GLOBALCONSTANTS PgnDef (* Global constants *)
  (* Standard: 61499-1 *)
  (* Version 1.0, 2026-06-29, Franz Höpfinger, Demmler Andreas Fahrzeugbau *)
  PACKAGE isobus::pgn::const;
  VAR_GLOBAL CONSTANT
    PGN_TORQUE_SPEED_CONTROL1 : UDINT := UDINT#16#0000; (* < 00000 - TSC1 *)
    PGN_TRANSMISSION_CONTROL1 : UDINT := UDINT#16#0100; (* < 00256 - TC1 *)
    PGN_ELECTRONIC_BRAKE_SYSTEM_1_1 : UDINT := UDINT#16#0200; (* < 00512 - EBS11 *)
    PGN_ELECTRONIC_BRAKE_SYSTEM_2_1 : UDINT := UDINT#16#0300; (* < 00768 - EBS21 *)
    PGN_EXTERNAL_BRAKE_REQUEST : UDINT := UDINT#16#0400; (* < 01024 - XBR *)
    PGN_CANOPEN_APPLICATION_MESSAGE_1_1 : UDINT := UDINT#16#0500; (* < 01280 - CAM11 *)
    PGN_CANOPEN_APPLICATION_MESSAGE_2_1 : UDINT := UDINT#16#0600; (* < 01536 - CAM21 *)
    PGN_GENERAL_PURPOSE_VALVE_PRESSURE : UDINT := UDINT#16#0700; (* < 01792 - GPV4 *)
    PGN_AUXILIARY_INPUT_OUTPUT_STATUS_5 : UDINT := UDINT#16#0800; (* < 02048 - AUXIO5 *)
    PGN_STATIC_ROLL_ANGLE_SENSOR_INFORMATION : UDINT := UDINT#16#0900; (* < 02304 - SRASI *)
    PGN_CRUISE_CONTROL_VEHICLE_SPEED_2 : UDINT := UDINT#16#0A00; (* < 02560 - CCVS2 *)
    PGN_ADVANCED_EMERGENCY_BRAKING_SYSTEM_2 : UDINT := UDINT#16#0B00; (* < 02816 - AEBS2 *)
    PGN_ELECTRONIC_ENGINE_CONTROLLER_16 : UDINT := UDINT#16#0C00; (* < 03072 - EEC16 *)
    PGN_TRANSMISSION_CONTROL_2 : UDINT := UDINT#16#0D00; (* < 03328 - TC2 *)
    PGN_SAFETY_HEADER_MESSAGE : UDINT := UDINT#16#0E00; (* < 03584 - SHM *)
    PGN_HIGH_VOLTAGE_ENERGY_STORAGE_PACK_11_CONTROL_1 : UDINT := UDINT#16#0F00; (* < 03840 - HVESP11C1 *)
    PGN_HIGH_VOLTAGE_ENERGY_STORAGE_PACK_12_CONTROL_1 : UDINT := UDINT#16#1000; (* < 04096 - HVESP12C1 *)
    PGN_HIGH_VOLTAGE_ENERGY_STORAGE_PACK_13_CONTROL_1 : UDINT := UDINT#16#1100; (* < 04352 - HVESP13C1 *)
    PGN_HIGH_VOLTAGE_ENERGY_STORAGE_PACK_14_CONTROL_1 : UDINT := UDINT#16#1200; (* < 04608 - HVESP14C1 *)
    PGN_HIGH_VOLTAGE_ENERGY_STORAGE_PACK_15_CONTROL_1 : UDINT := UDINT#16#1300; (* < 04864 - HVESP15C1 *)
    PGN_HIGH_VOLTAGE_ENERGY_STORAGE_PACK_16_CONTROL_1 : UDINT := UDINT#16#1400; (* < 05120 - HVESP16C1 *)
    PGN_HIGH_VOLTAGE_ENERGY_STORAGE_PACK_17_CONTROL_1 : UDINT := UDINT#16#1500; (* < 05376 - HVESP17C1 *)
    PGN_HIGH_VOLTAGE_ENERGY_STORAGE_PACK_18_CONTROL_1 : UDINT := UDINT#16#1600; (* < 05632 - HVESP18C1 *)
    PGN_HIGH_VOLTAGE_ENERGY_STORAGE_PACK_19_CONTROL_1 : UDINT := UDINT#16#1700; (* < 05888 - HVESP19C1 *)
    PGN_HIGH_VOLTAGE_ENERGY_STORAGE_PACK_20_CONTROL_1 : UDINT := UDINT#16#1800; (* < 06144 - HVESP20C1 *)
    PGN_HIGH_VOLTAGE_ENERGY_STORAGE_PACK_21_CONTROL_1 : UDINT := UDINT#16#1900; (* < 06400 - HVESP21C1 *)
    PGN_HIGH_VOLTAGE_ENERGY_STORAGE_PACK_22_CONTROL_1 : UDINT := UDINT#16#1A00; (* < 06656 - HVESP22C1 *)
    PGN_HIGH_VOLTAGE_ENERGY_STORAGE_SYSTEM_CONTROL_1 : UDINT := UDINT#16#1B00; (* < 06912 - HVESSC1 *)
    PGN_TRANSMISSION_CONTROL_3_OBSOLETE_SEE_PGN_16896 : UDINT := UDINT#16#1C00; (* < 07168 - TC3 *)
    PGN_ENGINE_IGNITION_CONTROLLER : UDINT := UDINT#16#1D00; (* < 07424 - EIC *)
    PGN_ALTERNATOR_CONTROL : UDINT := UDINT#16#1E00; (* < 07680 - ALTC *)
    PGN_HIGH_VOLTAGE_ENERGY_STORAGE_PACK_23_CONTROL_1 : UDINT := UDINT#16#1F00; (* < 07936 - HVESP23C1 *)
    PGN_HIGH_VOLTAGE_ENERGY_STORAGE_PACK_24_CONTROL_1 : UDINT := UDINT#16#2000; (* < 08192 - HVESP24C1 *)
    PGN_HIGH_VOLTAGE_ENERGY_STORAGE_PACK_25_CONTROL_1 : UDINT := UDINT#16#2100; (* < 08448 - HVESP25C1 *)
    PGN_HIGH_VOLTAGE_ENERGY_STORAGE_PACK_26_CONTROL_1 : UDINT := UDINT#16#2200; (* < 08704 - HVESP26C1 *)
    PGN_TIMS_TO_TIMC : UDINT := UDINT#16#2300; (* < 08960 - TIM12 *)
    PGN_TIMC_TO_TIMS : UDINT := UDINT#16#2400; (* < 09216 - TIM21 *)
    PGN_MULTI_PG : UDINT := UDINT#16#2500; (* < 09472 - MCPG *)
    PGN_MOTOR_GENERATOR_1_INVERTER_CONTROL : UDINT := UDINT#16#2600; (* < 09728 - MG1IC *)
    PGN_MOTOR_GENERATOR_2_INVERTER_CONTROL : UDINT := UDINT#16#2700; (* < 09984 - MG2IC *)
    PGN_MOTOR_GENERATOR_1_INVERTER_RATE_LIMITS_REQUEST_1 : UDINT := UDINT#16#2800; (* < 10240 - MG1IRLR1 *)
    PGN_MOTOR_GENERATOR_2_INVERTER_RATE_LIMITS_REQUEST_1 : UDINT := UDINT#16#2900; (* < 10496 - MG2IRLR1 *)
    PGN_HIGH_VOLTAGE_ENERGY_STORAGE_PACK_1_CONTROL_1 : UDINT := UDINT#16#2A00; (* < 10752 - HVESP1C1 *)
    PGN_HIGH_VOLTAGE_ENERGY_STORAGE_PACK_2_CONTROL_1 : UDINT := UDINT#16#2B00; (* < 11008 - HVESP2C1 *)
    PGN_HIGH_VOLTAGE_ENERGY_STORAGE_PACK_3_CONTROL_1 : UDINT := UDINT#16#2C00; (* < 11264 - HVESP3C1 *)
    PGN_HIGH_VOLTAGE_ENERGY_STORAGE_PACK_4_CONTROL_1 : UDINT := UDINT#16#2D00; (* < 11520 - HVESP4C1 *)
    PGN_HIGH_VOLTAGE_ENERGY_STORAGE_PACK_5_CONTROL_1 : UDINT := UDINT#16#2E00; (* < 11776 - HVESP5C1 *)
    PGN_HIGH_VOLTAGE_ENERGY_STORAGE_PACK_6_CONTROL_1 : UDINT := UDINT#16#2F00; (* < 12032 - HVESP6C1 *)
    PGN_HIGH_VOLTAGE_ENERGY_STORAGE_PACK_7_CONTROL_1 : UDINT := UDINT#16#3000; (* < 12288 - HVESP7C1 *)
    PGN_HIGH_VOLTAGE_ENERGY_STORAGE_PACK_8_CONTROL_1 : UDINT := UDINT#16#3100; (* < 12544 - HVESP8C1 *)
    PGN_HIGH_VOLTAGE_ENERGY_STORAGE_PACK_9_CONTROL_1 : UDINT := UDINT#16#3200; (* < 12800 - HVESP9C1 *)
    PGN_HIGH_VOLTAGE_ENERGY_STORAGE_PACK_10_CONTROL_1 : UDINT := UDINT#16#3300; (* < 13056 - HVESP10C1 *)
    PGN_RELIABLE_LONG_MESSAGE : UDINT := UDINT#16#3400; (* < 13312 - CJLFI *)
    PGN_RELIABLE_SHORT_MESSAGE : UDINT := UDINT#16#3500; (* < 13568 - CJSFWI *)
    PGN_UNRELIABLE_MESSAGE : UDINT := UDINT#16#3600; (* < 13824 - CJSFOI *)
    PGN_MESSAGE_ACKNOWLEDGEMENT : UDINT := UDINT#16#3700; (* < 14080 - CJCFI *)
    PGN_VERSION_NEGOTIATION_SECTION : UDINT := UDINT#16#3800; (* < 14336 - CJVGM *)
    PGN_EXTERNAL_ACC_ACCELERATION_REQUEST : UDINT := UDINT#16#3900; (* < 14592 - XAR *)
    PGN_BATTERY_CHARGER_1_COMMAND_1 : UDINT := UDINT#16#3A00; (* < 14848 - BCH1C1 *)
    PGN_BATTERY_CHARGER_2_COMMAND_1 : UDINT := UDINT#16#3B00; (* < 15104 - BCH2C1 *)
    PGN_TRACTOR_IMPLEMENT_MANAGEMENT_TIM_SERVER_TO_TIM_CLIENT_CONTROL_STATUS : UDINT := UDINT#16#3C00; (* < 15360 - TIM12_CS *)
    PGN_TRACTOR_IMPLEMENT_MANAGEMENT_TIM_CLIENT_TO_TIM_SERVER_CONTROL_STATUS : UDINT := UDINT#16#3D00; (* < 15616 - TIM21_CS *)
    PGN_FUEL_CELL_SYSTEM_CONTROL_COMMAND : UDINT := UDINT#16#3E00; (* < 15872 - FCSCC *)
    PGN_FUEL_CELL_SYSTEM_POWER_LIMIT_COMMAND : UDINT := UDINT#16#3F00; (* < 16128 - FCSPLC *)
    PGN_FUEL_CELL_SYSTEM_CURRENT_LIMIT_COMMAND : UDINT := UDINT#16#4000; (* < 16384 - FCSCLC *)
    PGN_HYDROGEN_STORAGE_SYSTEM_CONTROL_COMMAND : UDINT := UDINT#16#4100; (* < 16640 - HSSCC *)
    PGN_TRANSMISSION_CONTROL_4 : UDINT := UDINT#16#4200; (* < 16896 - TC4 *)
    PGN_SAFETY_HEADER_MESSAGE_2 : UDINT := UDINT#16#4300; (* < 17152 - SHM2 *)
    PGN_API_SELECT : UDINT := UDINT#16#4600; (* < 17920 - APISEL *)
    PGN_TRACTOR_IMPLEMENT_MANAGEMENT_TIM_SERVER_TO_CLIENT_INITIALIZATION_PARAMETE_X : UDINT := UDINT#16#4800; (* < 18432 - TIM12_IP *)
    PGN_TRACTOR_IMPLEMENT_MANAGEMENT_TIM_CLIENT_TO_SERVER_INITIALIZATION_PARAMETE_X : UDINT := UDINT#16#4900; (* < 18688 - TIM21_IP *)
    PGN_EV_MULTI_CONNECTION_DC_STATUS_1 : UDINT := UDINT#16#4A00; (* < 18944 - EVMCDCS1 *)
    PGN_EV_MULTI_CONNECTION_DC_CHARGING_LIMITS_1 : UDINT := UDINT#16#4B00; (* < 19200 - EVMCDCLIM1 *)
    PGN_ELECTRIFIED_ACCESSORY_ENGINE_COOLANT_PUMP_COMMAND : UDINT := UDINT#16#4C00; (* < 19456 - EAECPC *)
    PGN_FD_TRANSPORT_PROTOCOL_CONNECTION_MGMT : UDINT := UDINT#16#4D00; (* < 19712 - FD.TP.CM *)
    PGN_FD_TRANSPORT_PROTOCOL_DATA_TRANSFER : UDINT := UDINT#16#4E00; (* < 19968 - FD.TP.DT *)
    PGN_DATA_TRANSFER_SUPPORT : UDINT := UDINT#16#4F00; (* < 20224 - DTS *)
    PGN_MONTHLY_DATA_TRANSFER : UDINT := UDINT#16#5000; (* < 20480 - MDT *)
    PGN_WEEKLY_DATA_TRANSFER : UDINT := UDINT#16#5100; (* < 20736 - WDT *)
    PGN_DAILY_DATA_TRANSFER : UDINT := UDINT#16#5200; (* < 20992 - DDT *)
    PGN_EVSE_CONTROL_1 : UDINT := UDINT#16#5300; (* < 21248 - EVSEC1 *)
    PGN_WINCH_INFORMATION_3 : UDINT := UDINT#16#5400; (* < 21504 - WINCH3 *)
    PGN_AIR_SUSPENSION_CONTROL_8 : UDINT := UDINT#16#5500; (* < 21760 - ASC8 *)
    PGN_MOTOR_GENERATOR_2_INVERTER_CONTROL_2 : UDINT := UDINT#16#5600; (* < 22016 - MG2IC2 *)
    PGN_MOTOR_GENERATOR_1_INVERTER_CONTROL_2 : UDINT := UDINT#16#5700; (* < 22272 - MG1IC2 *)
    PGN_HOIST_COMMAND_INFORMATION : UDINT := UDINT#16#5800; (* < 22528 - HCI2 *)
    PGN_MOTOR_GENERATOR_2_INVERTER_ISOLATION_INTEGRITY_REQUEST : UDINT := UDINT#16#5900; (* < 22784 - MG2IIR *)
    PGN_MOTOR_GENERATOR_1_INVERTER_ISOLATION_INTEGRITY_REQUEST : UDINT := UDINT#16#5A00; (* < 23040 - MG1IIR *)
    PGN_MOTOR_GENERATOR_2_INVERTER_LIMITS_REQUEST_POWER : UDINT := UDINT#16#5B00; (* < 23296 - MG2IRP *)
    PGN_MOTOR_GENERATOR_2_INVERTER_LIMITS_REQUEST_MECHANICAL : UDINT := UDINT#16#5C00; (* < 23552 - MG2ILRM *)
    PGN_MOTOR_GENERATOR_2_INVERTER_LIMITS_REQUEST_DC_SIDE : UDINT := UDINT#16#5D00; (* < 23808 - MG2ILRDC *)
    PGN_MOTOR_GENERATOR_1_INVERTER_LIMITS_REQUEST_DC_SIDE : UDINT := UDINT#16#5E00; (* < 24064 - MG1ILRDC *)
    PGN_MOTOR_GENERATOR_1_INVERTER_LIMITS_REQUEST_MECHANICAL : UDINT := UDINT#16#5F00; (* < 24320 - MG1ILRM *)
    PGN_MOTOR_GENERATOR_1_INVERTER_LIMITS_REQUEST_POWER : UDINT := UDINT#16#6000; (* < 24576 - MG1IRP *)
    PGN_PERSONNEL_DETECT_INTERLOCK : UDINT := UDINT#16#6100; (* < 24832 - PDI *)
    PGN_ENGINE_CYLINDER_COMBUSTION_CONFIGURATION_FEEDBACK : UDINT := UDINT#16#6200; (* < 25088 - ECCCF *)
    PGN_ENGINE_CYLINDER_COMBUSTION_CONFIGURATION : UDINT := UDINT#16#6300; (* < 25344 - ECCC *)
    PGN_ENGINE_CYLINDER_PRESSURE_TIMING_FEEDBACK : UDINT := UDINT#16#6400; (* < 25600 - ECPTF *)
    PGN_ENGINE_CYLINDER_PRESSURE_TIMING_CONFIGURATION : UDINT := UDINT#16#6500; (* < 25856 - ECPTC *)
    PGN_ELECTRIFIED_ACCESSORY_GENERATOR_COOLANT_PUMP_COMMAND : UDINT := UDINT#16#6600; (* < 26112 - EAGCPC *)
    PGN_ELECTRIFIED_ACCESSORY_GENERATOR_COOLANT_FAN_COMMAND : UDINT := UDINT#16#6700; (* < 26368 - EAGCFC *)
    PGN_ON_BOARD_PROGRAMMING_1 : UDINT := UDINT#16#6800; (* < 26624 - OBP1 *)
    PGN_MARINE_CONTROL_INFORMATION_CONFIGURATION_1 : UDINT := UDINT#16#6900; (* < 26880 - MCIC1 *)
    PGN_MARINE_CONTROL_INFORMATION_2 : UDINT := UDINT#16#6A00; (* < 27136 - MCI2 *)
    PGN_WELL_STIMULATION_PUMP_SENSOR_CALIBRATION_COMMAND : UDINT := UDINT#16#6B00; (* < 27392 - WSPSCC *)
    PGN_CIA_602_2_XCP_OBSOLETE : UDINT := UDINT#16#6C00; (* < 27648 - CXCP *)
    PGN_WELL_STIMULATION_PUMP_SYSTEM_CONFIGURATION_COMMAND : UDINT := UDINT#16#6D00; (* < 27904 - WSPT1 *)
    PGN_CONFIGURABLE_RECEIVE_SPNS_COMMAND : UDINT := UDINT#16#6E00; (* < 28160 - CRSC *)
    PGN_AUTC_TO_AUTS : UDINT := UDINT#16#6F00; (* < 28416 - AUTH21 *)
    PGN_AUTS_TO_AUTC : UDINT := UDINT#16#7000; (* < 28672 - AUTH12 *)
    PGN_CONFIGURABLE_TRANSMIT_PGNS_COMMAND : UDINT := UDINT#16#7100; (* < 28928 - CTPC *)
    PGN_OIL_DEBRIS_MONITOR_CONFIGURATION_COMMAND : UDINT := UDINT#16#7200; (* < 29184 - ODMCC *)
    PGN_ELECTRIFIED_ACCESSORY_PROPULSION_MOTOR_COOLANT_FAN_3_COMMAND : UDINT := UDINT#16#7300; (* < 29440 - EAPMCF3C *)
    PGN_ELECTRIFIED_ACCESSORY_PROPULSION_MOTOR_COOLANT_FAN_2_COMMAND : UDINT := UDINT#16#7400; (* < 29696 - EAPMCF2C *)
    PGN_ELECTRIFIED_ACCESSORY_PROPULSION_MOTOR_COOLANT_FAN_1_COMMAND : UDINT := UDINT#16#7500; (* < 29952 - EAPMCF1C *)
    PGN_ELECTRIFIED_ACCESSORY_POWER_ELECTRONICS_COOLANT_FAN_3_COMMAND : UDINT := UDINT#16#7600; (* < 30208 - EAPECF3C *)
    PGN_ELECTRIFIED_ACCESSORY_POWER_ELECTRONICS_COOLANT_FAN_2_COMMAND : UDINT := UDINT#16#7700; (* < 30464 - EAPECF2C *)
    PGN_ELECTRIFIED_ACCESSORY_POWER_ELECTRONICS_COOLANT_FAN_1_COMMAND : UDINT := UDINT#16#7800; (* < 30720 - EAPECF1C *)
    PGN_ELECTRIFIED_ACCESSORY_PROPULSION_MOTOR_OIL_PUMP_COMMAND : UDINT := UDINT#16#7900; (* < 30976 - EAPMOPC *)
    PGN_ELECTRIFIED_ACCESSORY_PROPULSION_MOTOR_COOLANT_PUMP_COMMAND : UDINT := UDINT#16#7A00; (* < 31232 - EAPMCPC *)
    PGN_ELECTRIFIED_ACCESSORY_POWER_ELECTRONICS_COOLANT_PUMP_COMMAND : UDINT := UDINT#16#7B00; (* < 31488 - EAPECPC *)
    PGN_EXTENDED_CONTROL_FUNCTION_FUNCTIONALITIES : UDINT := UDINT#16#7C00; (* < 31744 - ECFF *)
    PGN_ELECTRIFIED_ACCESSORY_MOTOR_COMMAND : UDINT := UDINT#16#7D00; (* < 32000 - EAMC *)
    PGN_ENGINE_SPEED_RAMP_RATE_BOUNDARY_REQUEST : UDINT := UDINT#16#7E00; (* < 32256 - ESRRBR *)
    PGN_TIRE_SENSOR_IDENTIFICATION_COMMAND : UDINT := UDINT#16#7F00; (* < 32512 - TSIC *)
    PGN_HYBRID_OR_EV_SYSTEM_CONTROL_1 : UDINT := UDINT#16#8000; (* < 32768 - HSC1 *)
    PGN_AFTERTREATMENT_SYSTEM_CONTROL : UDINT := UDINT#16#8100; (* < 33024 - AFTSC *)
    PGN_TIRE_CONFIGURATION_COMMAND_INFORMATION : UDINT := UDINT#16#8200; (* < 33280 - TCCI *)
    PGN_PAYLOAD_CALIBRATION_INFORMATION_COMMAND : UDINT := UDINT#16#8300; (* < 33536 - PCIC *)
    PGN_AFTERTREATMENT_1_PARTICULATE_SENSOR_CONTROL : UDINT := UDINT#16#8400; (* < 33792 - AFT1PSC *)
    PGN_CAB_MESSAGE_2 : UDINT := UDINT#16#8500; (* < 34048 - CM2 *)
    PGN_SWITCHED_POWER_OUTPUTS_COMMAND : UDINT := UDINT#16#8600; (* < 34304 - SPOC *)
    PGN_ENGINE_STATE_REQUESTS : UDINT := UDINT#16#8700; (* < 34560 - ESR *)
    PGN_RADIO_BEACON_REQUEST : UDINT := UDINT#16#8800; (* < 34816 - RBR *)
    PGN_RUNNING_GEAR_EQUIPMENT_2_4 : UDINT := UDINT#16#8900; (* < 35072 - RGE24 *)
    PGN_RUNNING_GEAR_EQUIPMENT_1_2 : UDINT := UDINT#16#8A00; (* < 35328 - RGE12 *)
    PGN_CCP_DATA_TRANSMISSION_OBJECT : UDINT := UDINT#16#8B00; (* < 35584 - CCP_DTO *)
    PGN_CCP_COMMAND_RECEIVE_OBJECT : UDINT := UDINT#16#8C00; (* < 35840 - CCP_CRO *)
    PGN_SCC_TO_SCM : UDINT := UDINT#16#8D00; (* < 36096 - SCCCM *)
    PGN_SCM_TO_SCC : UDINT := UDINT#16#8E00; (* < 36352 - SCMCC *)
    PGN_ENGINE_CONFIGURATION_COMMANDS : UDINT := UDINT#16#8F00; (* < 36608 - ECC *)
    PGN_SUPPLEMENTAL_FAN_COMMAND : UDINT := UDINT#16#9000; (* < 36864 - SFC *)
    PGN_VEHICLE_CHASSIS_LUBRICATION_SYSTEM_1 : UDINT := UDINT#16#9100; (* < 37120 - VLS1 *)
    PGN_AFTERTREATMENT_1_HYDROCARBON_DOSER_INFORMATION_1 : UDINT := UDINT#16#9200; (* < 37376 - HCDI1 *)
    PGN_NAME_MANAGEMENT : UDINT := UDINT#16#9300; (* < 37632 - NM *)
    PGN_AFTERTREATMENT_1_DIESEL_PARTICULATE_FILTER_SOOT_SENSOR_CALIBRATION : UDINT := UDINT#16#9400; (* < 37888 - AT1DPFSSC *)
    PGN_AFTERTREATMENT_2_DIESEL_PARTICULATE_FILTER_SOOT_SENSOR_CALIBRATION : UDINT := UDINT#16#9500; (* < 38144 - AT2DPFSSC *)
    PGN_LOW_VOLTAGE_DISCONNECT_SET_OPERATING_MODE : UDINT := UDINT#16#9600; (* < 38400 - LVDSOM *)
    PGN_NOISE_CONTROL_STATUS : UDINT := UDINT#16#9700; (* < 38656 - NCS *)
    PGN_NOISE_CONTROL_1 : UDINT := UDINT#16#9800; (* < 38912 - NC1 *)
    PGN_JOYSTICK_LAMP_COMMAND_MESSAGE : UDINT := UDINT#16#9900; (* < 39168 - JLCM *)
    PGN_GENERAL_PURPOSE_MESSAGE_1_8 : UDINT := UDINT#16#9A00; (* < 39424 - GPM18 *)
    PGN_PROPRIETARY_METHOD_IDENTIFICATION : UDINT := UDINT#16#9B00; (* < 39680 - PMI *)
    PGN_AUXILIARY_INPUT_OUTPUT_STATUS_7 : UDINT := UDINT#16#9C00; (* < 39936 - AUXIO7 *)
    PGN_AUXILIARY_INPUT_OUTPUT_STATUS_6 : UDINT := UDINT#16#9D00; (* < 40192 - AUXIO6 *)
    PGN_DTC_COUNTS : UDINT := UDINT#16#9E00; (* < 40448 - DM29 *)
    PGN_IMMEDIATE_FAULT_STATUS : UDINT := UDINT#16#9F00; (* < 40704 - DM35 *)
    PGN_NTE_STATUS : UDINT := UDINT#16#A000; (* < 40960 - DM34 *)
    PGN_EMISSION_INCREASING_AUXILIARY_EMISSION_CONTROL_DEVICE_ACTIVE_TIME : UDINT := UDINT#16#A100; (* < 41216 - DM33 *)
    PGN_REGULATED_EXHAUST_EMISSION_LEVEL_EXCEEDANCE : UDINT := UDINT#16#A200; (* < 41472 - DM32 *)
    PGN_DTC_TO_LAMP_ASSOCIATION : UDINT := UDINT#16#A300; (* < 41728 - DM31 *)
    PGN_SCALED_TEST_RESULTS : UDINT := UDINT#16#A400; (* < 41984 - DM30 *)
    PGN_AUXILIARY_INPUT_OUTPUT_STATUS_4 : UDINT := UDINT#16#A500; (* < 42240 - AUXIO4 *)
    PGN_AUXILIARY_INPUT_OUTPUT_STATUS_3 : UDINT := UDINT#16#A600; (* < 42496 - AUXIO3 *)
    PGN_AUX_IO_STATUS_2 : UDINT := UDINT#16#A700; (* < 42752 - AUXIO2 *)
    PGN_TEXT_DISPLAY : UDINT := UDINT#16#A800; (* < 43008 - DISP1 *)
    PGN_FORWARD_LANE_IMAGE_COMMAND : UDINT := UDINT#16#A900; (* < 43264 - FLIC *)
    PGN_FSC_TO_FS : UDINT := UDINT#16#AA00; (* < 43520 - CFS *)
    PGN_FS_TO_FSC : UDINT := UDINT#16#AB00; (* < 43776 - FSC *)
    PGN_GUIDANCE_MACHINE_STATUS : UDINT := UDINT#16#AC00; (* < 44032 - GMS *)
    PGN_GUIDANCE_SYSTEM_COMMAND_MSG : UDINT := UDINT#16#AD00; (* < 44288 - GSC *)
    PGN_TIRE_PRESSURE_REFERENCE_SETTING : UDINT := UDINT#16#AE00; (* < 44544 - TPRS *)
    PGN_PARAMETER_LOCATE_MESSAGE : UDINT := UDINT#16#AF00; (* < 44800 - PLM *)
    PGN_CONFIGURATION_IDENTIFICATION_MESSAGE : UDINT := UDINT#16#B000; (* < 45056 - CIM *)
    PGN_PROPRIETARILY_CONFIGURABLE_MESSAGE_1 : UDINT := UDINT#16#B100; (* < 45312 - PCM1 *)
    PGN_PROPRIETARILY_CONFIGURABLE_MESSAGE_2 : UDINT := UDINT#16#B200; (* < 45568 - PCM2 *)
    PGN_PROPRIETARILY_CONFIGURABLE_MESSAGE_3 : UDINT := UDINT#16#B300; (* < 45824 - PCM3 *)
    PGN_PROPRIETARILY_CONFIGURABLE_MESSAGE_4 : UDINT := UDINT#16#B400; (* < 46080 - PCM4 *)
    PGN_PROPRIETARILY_CONFIGURABLE_MESSAGE_5 : UDINT := UDINT#16#B500; (* < 46336 - PCM5 *)
    PGN_PROPRIETARILY_CONFIGURABLE_MESSAGE_6 : UDINT := UDINT#16#B600; (* < 46592 - PCM6 *)
    PGN_PROPRIETARILY_CONFIGURABLE_MESSAGE_7 : UDINT := UDINT#16#B700; (* < 46848 - PCM7 *)
    PGN_PROPRIETARILY_CONFIGURABLE_MESSAGE_8 : UDINT := UDINT#16#B800; (* < 47104 - PCM8 *)
    PGN_PROPRIETARILY_CONFIGURABLE_MESSAGE_9 : UDINT := UDINT#16#B900; (* < 47360 - PCM9 *)
    PGN_PROPRIETARILY_CONFIGURABLE_MESSAGE_10 : UDINT := UDINT#16#BA00; (* < 47616 - PCM10 *)
    PGN_PROPRIETARILY_CONFIGURABLE_MESSAGE_11 : UDINT := UDINT#16#BB00; (* < 47872 - PCM11 *)
    PGN_PROPRIETARILY_CONFIGURABLE_MESSAGE_12 : UDINT := UDINT#16#BC00; (* < 48128 - PCM12 *)
    PGN_PROPRIETARILY_CONFIGURABLE_MESSAGE_13 : UDINT := UDINT#16#BD00; (* < 48384 - PCM13 *)
    PGN_PROPRIETARILY_CONFIGURABLE_MESSAGE_14 : UDINT := UDINT#16#BE00; (* < 48640 - PCM14 *)
    PGN_PROPRIETARILY_CONFIGURABLE_MESSAGE_15 : UDINT := UDINT#16#BF00; (* < 48896 - PCM15 *)
    PGN_PROPRIETARILY_CONFIGURABLE_MESSAGE_16 : UDINT := UDINT#16#C000; (* < 49152 - PCM16 *)
    PGN_DIAGNOSTIC_READINESS_2 : UDINT := UDINT#16#C100; (* < 49408 - DM21 *)
    PGN_MONITOR_PERFORMANCE_RATIO : UDINT := UDINT#16#C200; (* < 49664 - DM20 *)
    PGN_INDIVIDUAL_CLEAR_RESET_OF_ACTIVE_AND_PREVIOUSLY_ACTIVE_DTC : UDINT := UDINT#16#C300; (* < 49920 - DM22 *)
    PGN_GENPURPOSE_VALVE_COMMAND : UDINT := UDINT#16#C400; (* < 50176 - GPV3 *)
    PGN_GENPURPOSE_VALVE_MEASFLOW : UDINT := UDINT#16#C500; (* < 50432 - GPV2 *)
    PGN_GENPURPOSE_VALVE_ESTIMFLOW : UDINT := UDINT#16#C600; (* < 50688 - GPV1 *)
    PGN_ETP_DT : UDINT := UDINT#16#C700; (* < 50944 - ETP.DT *)
    PGN_ETP_CM : UDINT := UDINT#16#C800; (* < 51200 - ETP.CM *)
    PGN_REQUEST2_PGN : UDINT := UDINT#16#C900; (* < 51456 - RQST2 *)
    PGN_TRANSFER_PGN : UDINT := UDINT#16#CA00; (* < 51712 - XFER *)
    PGN_PROCESS_DATA : UDINT := UDINT#16#CB00; (* < 51968 - PD *)
    PGN_REQ_FOR_REP_RATE : UDINT := UDINT#16#CC00; (* < 52224 - REQRR *)
    PGN_DoCAN_MIXED_FUNCTIONAL : UDINT := UDINT#16#CD00; (* < 52480 - DIAG1 *)
    PGN_DoCAN_MIXED_PHYSICAL : UDINT := UDINT#16#CE00; (* < 52736 - DIAG2 *)
    PGN_CONTINUOUSTORQUE : UDINT := UDINT#16#CF00; (* < 52992 - CTL *)
    PGN_CAB_ILLUMINATION : UDINT := UDINT#16#D000; (* < 53248 - CL *)
    PGN_AIRSUSPENSION_CONTROL6 : UDINT := UDINT#16#D100; (* < 53504 - ASC6 *)
    PGN_AIRSUSPENSION_CONTROL2 : UDINT := UDINT#16#D200; (* < 53760 - ASC2 *)
    PGN_CALIBRATION_INFORMATION : UDINT := UDINT#16#D300; (* < 54016 - DM19 *)
    PGN_DATA_SECURITY_54272 : UDINT := UDINT#16#D400; (* < 54272 - DM18 *)
    PGN_DATA_SECURITY : UDINT := UDINT#16#D500; (* < 54528 - TDA *)
    PGN_BOOT_LOAD_DATA : UDINT := UDINT#16#D600; (* < 54784 - DM17 *)
    PGN_BINARY_DATA_TRANSFER : UDINT := UDINT#16#D700; (* < 55040 - DM16 *)
    PGN_MEMORY_ACCESS_RESPONSE : UDINT := UDINT#16#D800; (* < 55296 - DM15 *)
    PGN_MEMORY_ACCESS_REQUEST : UDINT := UDINT#16#D900; (* < 55552 - DM14 *)
    PGN_DoCAN_NORMAL_PHYSICAL : UDINT := UDINT#16#DA00; (* < 55808 - DIAG3 *)
    PGN_DoCAN_NORMAL_FUNCTIONAL : UDINT := UDINT#16#DB00; (* < 56064 - DIAG4 *)
    PGN_ANTI_SHEFT_STATUS : UDINT := UDINT#16#DC00; (* < 56320 - ATS *)
    PGN_ANTI_SHEFT_REQUEST : UDINT := UDINT#16#DD00; (* < 56576 - ATR *)
    PGN_RESET : UDINT := UDINT#16#DE00; (* < 56832 - RESET *)
    PGN_STOP_START_BROADCAST : UDINT := UDINT#16#DF00; (* < 57088 - DM13 *)
    PGN_CAB_MESSAGE1 : UDINT := UDINT#16#E000; (* < 57344 - CM1 *)
    PGN_GENERAL_PURPOSE_MESSAGE_2_1 : UDINT := UDINT#16#E100; (* < 57600 - GPM21 *)
    PGN_GENERAL_PURPOSE_MESSAGE_1_1 : UDINT := UDINT#16#E200; (* < 57856 - GPM11 *)
    PGN_CMD_NONCONTIN_MONITOR : UDINT := UDINT#16#E300; (* < 58112 - DM7 *)
    PGN_RUNNING_GEAR_EQUIPMENT_1_1 : UDINT := UDINT#16#E400; (* < 58368 - RGE11 *)
    PGN_RUNNING_GEAR_EQUIPMENT_2_1 : UDINT := UDINT#16#E500; (* < 58624 - RGE21 *)
    PGN_VTtoECU : UDINT := UDINT#16#E600; (* < 58880 - VT12 *)
    PGN_ECUtoVT : UDINT := UDINT#16#E700; (* < 59136 - VT21 *)
    PGN_N_ACK : UDINT := UDINT#16#E800; (* < 59392 - ACKM *)
    PGN_REQUEST_PGN : UDINT := UDINT#16#EA00; (* < 59904 - RQST *)
    PGN_TP_DT : UDINT := UDINT#16#EB00; (* < 60160 - TP.DT *)
    PGN_TP_CM : UDINT := UDINT#16#EC00; (* < 60416 - TP.CM.xx *)
    PGN_NETWORK_LAYER : UDINT := UDINT#16#ED00; (* < 60672 - N.xx *)
    PGN_ADDRESS_CLAIMED : UDINT := UDINT#16#EE00; (* < 60928 - AC *)
    PGN_CANNOT_CLAIM_SA : UDINT := UDINT#16#EE00; (* < 60928 - AC *)
    PGN_PDU1_PropA : UDINT := UDINT#16#EF00; (* < 61184 - PropA *)
    PGN_PDU2_240_X : UDINT := UDINT#16#F000; (* < 61440 - ERC1 *)
    PGN_ELEC_RETARDER_CONTROLLER : UDINT := UDINT#16#F000; (* < 61440 - ERC1 *)
    PGN_ELEC_BRAKE_CONTROLLER : UDINT := UDINT#16#F001; (* < 61441 - EBC1 *)
    PGN_ELEC_TRANSMISS_CONTROLLER_1 : UDINT := UDINT#16#F002; (* < 61442 - ETC1 *)
    PGN_ELEC_ENGINE_CONTROLLER_2 : UDINT := UDINT#16#F003; (* < 61443 - EEC2 *)
    PGN_ELEC_ENGINE_CONTROLLER_1 : UDINT := UDINT#16#F004; (* < 61444 - EEC1 *)
    PGN_ELEC_TRANSMISS_CONTROLLER_2 : UDINT := UDINT#16#F005; (* < 61445 - ETC2 *)
    PGN_ELEC_AXLE_CONTROLLER_1 : UDINT := UDINT#16#F006; (* < 61446 - EAC1 *)
    PGN_FORW_LANE_IMAGE_URGENT_MSG : UDINT := UDINT#16#F007; (* < 61447 - FLI1 *)
    PGN_HYDRAULIC_PRESS_GOVER_INFO : UDINT := UDINT#16#F008; (* < 61448 - HPG *)
    PGN_VEHICLE_DYN_STAB_CTRL_2 : UDINT := UDINT#16#F009; (* < 61449 - VDC2 *)
    PGN_ENGINE_GAS_FLOW_RATE : UDINT := UDINT#16#F00A; (* < 61450 - EGF1 *)
    PGN_ELECTRONIC_STEERING_CONTROL : UDINT := UDINT#16#F00B; (* < 61451 - ESC1 *)
    PGN_ELECTRONIC_TRANSMISSION_CONTROLLER_8 : UDINT := UDINT#16#F00C; (* < 61452 - ETC8 *)
    PGN_LAND_LEVELING_SYSTEM_OPERATIONAL_INFORMATION : UDINT := UDINT#16#F00D; (* < 61453 - LOI *)
    PGN_AFTERTREATMENT_1_INTAKE_GAS_1 : UDINT := UDINT#16#F00E; (* < 61454 - AT1IG1 *)
    PGN_AFTERTREATMENT_1_OUTLET_GAS_1 : UDINT := UDINT#16#F00F; (* < 61455 - AT1OG1 *)
    PGN_AFTERTREATMENT_2_INTAKE_GAS_1 : UDINT := UDINT#16#F010; (* < 61456 - AT2IG1 *)
    PGN_AFTERTREATMENT_2_OUTLET_GAS_1 : UDINT := UDINT#16#F011; (* < 61457 - AT2OG1 *)
    PGN_FIFTH_WHEEL_SMART_SYSTEMS_1 : UDINT := UDINT#16#F012; (* < 61458 - FWSS1 *)
    PGN_SLOPE_SENSOR_INFORMATION : UDINT := UDINT#16#F013; (* < 61459 - SSI *)
    PGN_BLADE_INFORMATION : UDINT := UDINT#16#F014; (* < 61460 - BI *)
    PGN_REQUESTED_GENERATOR_TOTAL_AC_REACTIVE_POWER : UDINT := UDINT#16#F015; (* < 61461 - RGTACRP *)
    PGN_CYLINDER_COMBUSTION_STATUS : UDINT := UDINT#16#F016; (* < 61462 - CCS *)
    PGN_ENGINE_KNOCK_LEVEL_1 : UDINT := UDINT#16#F017; (* < 61463 - KL1 *)
    PGN_ENGINE_KNOCK_LEVEL_2 : UDINT := UDINT#16#F018; (* < 61464 - KL2 *)
    PGN_ENGINE_KNOCK_LEVEL_3 : UDINT := UDINT#16#F019; (* < 61465 - KL3 *)
    PGN_ENGINE_THROTTLE_FUEL_ACTUATOR_CONTROL_COMMAND : UDINT := UDINT#16#F01A; (* < 61466 - TFAC *)
    PGN_GENERAL_PURPOSE_MESSAGE_1_7 : UDINT := UDINT#16#F01B; (* < 61467 - GPM17 *)
    PGN_REQUESTED_GENERATOR_AVERAGE_BASIC_AC_QUANTITIES : UDINT := UDINT#16#F01C; (* < 61468 - RGAAC *)
    PGN_STEERING_ANGLE_SENSOR_INFORMATION : UDINT := UDINT#16#F01D; (* < 61469 - SAS *)
    PGN_GENERATOR_CONTROL_2 : UDINT := UDINT#16#F01E; (* < 61470 - GC2 *)
    PGN_ELECTRONIC_BRAKE_SYSTEM_2_6 : UDINT := UDINT#16#F01F; (* < 61471 - EBS26 *)
    PGN_ELECTRONIC_BRAKE_SYSTEM_2_5 : UDINT := UDINT#16#F020; (* < 61472 - EBS25 *)
    PGN_ENGINE_SPEED_SENSOR_INFORMATION_1 : UDINT := UDINT#16#F021; (* < 61473 - ESSI1 *)
    PGN_MACHINE_SELECTED_SPEED : UDINT := UDINT#16#F022; (* < 61474 - MSS *)
    PGN_AFTERTREATMENT_1_SCR_DOSING_SYSTEM_INFORMATION_1 : UDINT := UDINT#16#F023; (* < 61475 - A1SCRDSI1 *)
    PGN_AFTERTREATMENT_1_SCR_DOSING_SYSTEM_REQUESTS_1 : UDINT := UDINT#16#F024; (* < 61476 - A1SCRDSR1 *)
    PGN_AFTERTREATMENT_1_SCR_AMMONIA_INFORMATION : UDINT := UDINT#16#F025; (* < 61477 - A1SCRAI *)
    PGN_AFTERTREATMENT_2_SCR_DOSING_SYSTEM_INFORMATION_1 : UDINT := UDINT#16#F026; (* < 61478 - A2SCRDSI1 *)
    PGN_AFTERTREATMENT_2_SCR_DOSING_SYSTEM_REQUESTS_1 : UDINT := UDINT#16#F027; (* < 61479 - A2SCRDSR1 *)
    PGN_AFTERTREATMENT_2_SCR_AMMONIA_INFORMATION : UDINT := UDINT#16#F028; (* < 61480 - A2SCRAI *)
    PGN_SLOPE_SENSOR_INFORMATION_2 : UDINT := UDINT#16#F029; (* < 61481 - SSI2 *)
    PGN_ANGULAR_RATE_INFORMATION : UDINT := UDINT#16#F02A; (* < 61482 - ARI *)
    PGN_CRASH_NOTIFICATION : UDINT := UDINT#16#F02B; (* < 61483 - CN *)
    PGN_MAGNET_STATUS_INFORMATION_2 : UDINT := UDINT#16#F02C; (* < 61484 - MSI2 *)
    PGN_ACCELERATION_SENSOR : UDINT := UDINT#16#F02D; (* < 61485 - ACCS *)
    PGN_ENGINE_TURBOCHARGER_CONTROL_1 : UDINT := UDINT#16#F02E; (* < 61486 - ETCC1 *)
    PGN_ADVANCED_EMERGENCY_BRAKING_SYSTEM_1 : UDINT := UDINT#16#F02F; (* < 61487 - AEBS1 *)
    PGN_WIRELESS_STATUS : UDINT := UDINT#16#F030; (* < 61488 - WS *)
    PGN_WAND_SENSOR : UDINT := UDINT#16#F031; (* < 61489 - WAND *)
    PGN_LINEAR_DISPLACEMENT_SENSOR : UDINT := UDINT#16#F032; (* < 61490 - LDISP *)
    PGN_AFTERTREATMENT_1_SCR_AMMONIA_INFORMATION_2 : UDINT := UDINT#16#F033; (* < 61491 - A1SCRAI2 *)
    PGN_AFTERTREATMENT_2_SCR_AMMONIA_INFORMATION_2 : UDINT := UDINT#16#F034; (* < 61492 - A2SCRAI2 *)
    PGN_HIGH_VOLTAGE_ENERGY_STORAGE_SYSTEM_STATUS_2 : UDINT := UDINT#16#F036; (* < 61494 - HVESSS2 *)
    PGN_ENGINE_TURBOCHARGER_BLOWOFF_ACTUATOR_1 : UDINT := UDINT#16#F037; (* < 61495 - ETBA1 *)
    PGN_ENGINE_TORQUE_FUEL_REQUEST : UDINT := UDINT#16#F038; (* < 61496 - ETFR *)
    PGN_ENGINE_AIR_SYSTEM_INFORMATION : UDINT := UDINT#16#F039; (* < 61497 - EASI *)
    PGN_ENGINE_CYLINDER_1_COMBUSTION_INFORMATION : UDINT := UDINT#16#F03A; (* < 61498 - ECCI1 *)
    PGN_ENGINE_CYLINDER_2_COMBUSTION_INFORMATION : UDINT := UDINT#16#F03B; (* < 61499 - ECCI2 *)
    PGN_ENGINE_CYLINDER_3_COMBUSTION_INFORMATION : UDINT := UDINT#16#F03C; (* < 61500 - ECCI3 *)
    PGN_ENGINE_CYLINDER_4_COMBUSTION_INFORMATION : UDINT := UDINT#16#F03D; (* < 61501 - ECCI4 *)
    PGN_ENGINE_CYLINDER_5_COMBUSTION_INFORMATION : UDINT := UDINT#16#F03E; (* < 61502 - ECCI5 *)
    PGN_ENGINE_CYLINDER_6_COMBUSTION_INFORMATION : UDINT := UDINT#16#F03F; (* < 61503 - ECCI6 *)
    PGN_ENGINE_CYLINDER_7_COMBUSTION_INFORMATION : UDINT := UDINT#16#F040; (* < 61504 - ECCI7 *)
    PGN_ENGINE_CYLINDER_8_COMBUSTION_INFORMATION : UDINT := UDINT#16#F041; (* < 61505 - ECCI8 *)
    PGN_ENGINE_CYLINDER_9_COMBUSTION_INFORMATION : UDINT := UDINT#16#F042; (* < 61506 - ECCI9 *)
    PGN_ENGINE_CYLINDER_10_COMBUSTION_INFORMATION : UDINT := UDINT#16#F043; (* < 61507 - ECCI10 *)
    PGN_ENGINE_CYLINDER_11_COMBUSTION_INFORMATION : UDINT := UDINT#16#F044; (* < 61508 - ECCI11 *)
    PGN_ENGINE_CYLINDER_12_COMBUSTION_INFORMATION : UDINT := UDINT#16#F045; (* < 61509 - ECCI12 *)
    PGN_ENGINE_CYLINDER_13_COMBUSTION_INFORMATION : UDINT := UDINT#16#F046; (* < 61510 - ECCI13 *)
    PGN_ENGINE_CYLINDER_14_COMBUSTION_INFORMATION : UDINT := UDINT#16#F047; (* < 61511 - ECCI14 *)
    PGN_ENGINE_CYLINDER_15_COMBUSTION_INFORMATION : UDINT := UDINT#16#F048; (* < 61512 - ECCI15 *)
    PGN_ENGINE_CYLINDER_16_COMBUSTION_INFORMATION : UDINT := UDINT#16#F049; (* < 61513 - ECCI16 *)
    PGN_ENGINE_CYLINDER_17_COMBUSTION_INFORMATION : UDINT := UDINT#16#F04A; (* < 61514 - ECCI17 *)
    PGN_ENGINE_CYLINDER_18_COMBUSTION_INFORMATION : UDINT := UDINT#16#F04B; (* < 61515 - ECCI18 *)
    PGN_ENGINE_CYLINDER_19_COMBUSTION_INFORMATION : UDINT := UDINT#16#F04C; (* < 61516 - ECCI19 *)
    PGN_ENGINE_CYLINDER_20_COMBUSTION_INFORMATION : UDINT := UDINT#16#F04D; (* < 61517 - ECCI20 *)
    PGN_ENGINE_CYLINDER_1_COMBUSTION_AVERAGE_INFORMATION : UDINT := UDINT#16#F04E; (* < 61518 - ECCAI1 *)
    PGN_ENGINE_CYLINDER_2_COMBUSTION_AVERAGE_INFORMATION : UDINT := UDINT#16#F04F; (* < 61519 - ECCAI2 *)
    PGN_ENGINE_CYLINDER_3_COMBUSTION_AVERAGE_INFORMATION : UDINT := UDINT#16#F050; (* < 61520 - ECCAI3 *)
    PGN_ENGINE_CYLINDER_4_COMBUSTION_AVERAGE_INFORMATION : UDINT := UDINT#16#F051; (* < 61521 - ECCAI4 *)
    PGN_ENGINE_CYLINDER_5_COMBUSTION_AVERAGE_INFORMATION : UDINT := UDINT#16#F052; (* < 61522 - ECCAI5 *)
    PGN_ENGINE_CYLINDER_6_COMBUSTION_AVERAGE_INFORMATION : UDINT := UDINT#16#F053; (* < 61523 - ECCAI6 *)
    PGN_ENGINE_CYLINDER_7_COMBUSTION_AVERAGE_INFORMATION : UDINT := UDINT#16#F054; (* < 61524 - ECCAI7 *)
    PGN_ENGINE_CYLINDER_8_COMBUSTION_AVERAGE_INFORMATION : UDINT := UDINT#16#F055; (* < 61525 - ECCAI8 *)
    PGN_ENGINE_CYLINDER_9_COMBUSTION_AVERAGE_INFORMATION : UDINT := UDINT#16#F056; (* < 61526 - ECCAI9 *)
    PGN_ENGINE_CYLINDER_10_COMBUSTION_AVERAGE_INFORMATION : UDINT := UDINT#16#F057; (* < 61527 - ECCAI10 *)
    PGN_ENGINE_CYLINDER_11_COMBUSTION_AVERAGE_INFORMATION : UDINT := UDINT#16#F058; (* < 61528 - ECCAI11 *)
    PGN_ENGINE_CYLINDER_12_COMBUSTION_AVERAGE_INFORMATION : UDINT := UDINT#16#F059; (* < 61529 - ECCAI12 *)
    PGN_ENGINE_CYLINDER_13_COMBUSTION_AVERAGE_INFORMATION : UDINT := UDINT#16#F05A; (* < 61530 - ECCAI13 *)
    PGN_ENGINE_CYLINDER_14_COMBUSTION_AVERAGE_INFORMATION : UDINT := UDINT#16#F05B; (* < 61531 - ECCAI14 *)
    PGN_ENGINE_CYLINDER_15_COMBUSTION_AVERAGE_INFORMATION : UDINT := UDINT#16#F05C; (* < 61532 - ECCAI15 *)
    PGN_ENGINE_CYLINDER_16_COMBUSTION_AVERAGE_INFORMATION : UDINT := UDINT#16#F05D; (* < 61533 - ECCAI16 *)
    PGN_ENGINE_CYLINDER_17_COMBUSTION_AVERAGE_INFORMATION : UDINT := UDINT#16#F05E; (* < 61534 - ECCAI17 *)
    PGN_ENGINE_CYLINDER_18_COMBUSTION_AVERAGE_INFORMATION : UDINT := UDINT#16#F05F; (* < 61535 - ECCAI18 *)
    PGN_ENGINE_CYLINDER_19_COMBUSTION_AVERAGE_INFORMATION : UDINT := UDINT#16#F060; (* < 61536 - ECCAI19 *)
    PGN_ENGINE_CYLINDER_20_COMBUSTION_AVERAGE_INFORMATION : UDINT := UDINT#16#F061; (* < 61537 - ECCAI20 *)
    PGN_ELECTRONIC_TRANSMISSION_CONTROLLER_12 : UDINT := UDINT#16#F062; (* < 61538 - ETC12 *)
    PGN_FUEL_INFORMATION_5_GASEOUS : UDINT := UDINT#16#F063; (* < 61539 - GFI5 *)
    PGN_ENGINE_GASEOUS_FUEL_VALVE_DURATION_COMMAND_1 : UDINT := UDINT#16#F064; (* < 61540 - EGFVDC1 *)
    PGN_ENGINE_GASEOUS_FUEL_VALVE_DURATION_COMMAND_2 : UDINT := UDINT#16#F065; (* < 61541 - EGFVDC2 *)
    PGN_ENGINE_GASEOUS_FUEL_VALVE_DURATION_COMMAND_3 : UDINT := UDINT#16#F066; (* < 61542 - EGFVDC3 *)
    PGN_ENGINE_GASEOUS_FUEL_VALVE_DURATION_COMMAND_4 : UDINT := UDINT#16#F067; (* < 61543 - EGFVDC4 *)
    PGN_ENGINE_GASEOUS_FUEL_VALVE_DURATION_COMMAND_5 : UDINT := UDINT#16#F068; (* < 61544 - EGFVDC5 *)
    PGN_ENGINE_GASEOUS_FUEL_VALVE_START_OF_ACTUATION_COMMAND_1 : UDINT := UDINT#16#F069; (* < 61545 - EGFVSOAC1 *)
    PGN_ENGINE_GASEOUS_FUEL_VALVE_START_OF_ACTUATION_COMMAND_2 : UDINT := UDINT#16#F06A; (* < 61546 - EGFVSOAC2 *)
    PGN_ENGINE_GASEOUS_FUEL_VALVE_START_OF_ACTUATION_COMMAND_3 : UDINT := UDINT#16#F06B; (* < 61547 - EGFVSOAC3 *)
    PGN_ENGINE_GASEOUS_FUEL_VALVE_START_OF_ACTUATION_COMMAND_4 : UDINT := UDINT#16#F06C; (* < 61548 - EGFVSOAC4 *)
    PGN_ENGINE_GASEOUS_FUEL_VALVE_START_OF_ACTUATION_COMMAND_5 : UDINT := UDINT#16#F06D; (* < 61549 - EGFVSOAC5 *)
    PGN_FUEL_PUMP_ACTUATOR_CONTROL_COMMAND : UDINT := UDINT#16#F06E; (* < 61550 - FPAC *)
    PGN_POWER_CONVERTER_1_CONTROL_1 : UDINT := UDINT#16#F06F; (* < 61551 - PC1IC1 *)
    PGN_POWER_CONVERTER_2_CONTROL_1 : UDINT := UDINT#16#F070; (* < 61552 - PC2IC1 *)
    PGN_POWER_CONVERTER_1_RATE_LIMITS_REQUEST_1 : UDINT := UDINT#16#F071; (* < 61553 - PC1IRLR1 *)
    PGN_POWER_CONVERTER_2_RATE_LIMITS_REQUEST_1 : UDINT := UDINT#16#F072; (* < 61554 - PC2IRLR1 *)
    PGN_POWER_CONVERTER_2_CONTROL_2 : UDINT := UDINT#16#F073; (* < 61555 - PC2IC2 *)
    PGN_POWER_CONVERTER_1_CONTROL_2 : UDINT := UDINT#16#F074; (* < 61556 - PC1IC2 *)
    PGN_POWER_CONVERTER_1_MODE_FEEDBACK_1 : UDINT := UDINT#16#F075; (* < 61557 - PC1IMF1 *)
    PGN_POWER_CONVERTER_1_LIMITS_ACTIVE_POWER : UDINT := UDINT#16#F076; (* < 61558 - PC1ILAP *)
    PGN_POWER_CONVERTER_1_LIMITS_ACTIVE_ELECTRICAL : UDINT := UDINT#16#F077; (* < 61559 - PC1ILAM *)
    PGN_POWER_CONVERTER_1_LIMITS_ACTIVE_DC_ENERGY_SOURCE_1 : UDINT := UDINT#16#F078; (* < 61560 - PC1ILADC *)
    PGN_POWER_CONVERTER_1_LOW_VOLTAGE : UDINT := UDINT#16#F079; (* < 61561 - PC1ILV *)
    PGN_POWER_CONVERTER_2_MODE_FEEDBACK_1 : UDINT := UDINT#16#F07A; (* < 61562 - PC2IMF1 *)
    PGN_POWER_CONVERTER_2_LIMITS_ACTIVE_POWER : UDINT := UDINT#16#F07B; (* < 61563 - PC2ILAP *)
    PGN_POWER_CONVERTER_2_LIMITS_ACTIVE_ELECTRICAL : UDINT := UDINT#16#F07C; (* < 61564 - PC2ILAM *)
    PGN_POWER_CONVERTER_2_LIMITS_ACTIVE_DC_ENERGY_SOURCE_1 : UDINT := UDINT#16#F07D; (* < 61565 - PC2ILADC *)
    PGN_POWER_CONVERTER_2_LOW_VOLTAGE : UDINT := UDINT#16#F07E; (* < 61566 - PC2ILV *)
    PGN_POWER_CONVERTER_1_STATUS_2 : UDINT := UDINT#16#F07F; (* < 61567 - PC1IS2 *)
    PGN_POWER_CONVERTER_1_RATE_LIMITS_ACTIVE_1 : UDINT := UDINT#16#F080; (* < 61568 - PC1IRLA1 *)
    PGN_POWER_CONVERTER_2_STATUS_2 : UDINT := UDINT#16#F081; (* < 61569 - PC2IS2 *)
    PGN_POWER_CONVERTER_2_RATE_LIMITS_ACTIVE_1 : UDINT := UDINT#16#F082; (* < 61570 - PC2IRLA1 *)
    PGN_POWER_CONVERTER_2_ISOLATION_INTEGRITY : UDINT := UDINT#16#F083; (* < 61571 - PC2II *)
    PGN_POWER_CONVERTER_1_ISOLATION_INTEGRITY : UDINT := UDINT#16#F084; (* < 61572 - PC1II *)
    PGN_POWER_CONVERTER_2_STATUS_1 : UDINT := UDINT#16#F085; (* < 61573 - PC2IS1 *)
    PGN_POWER_CONVERTER_1_STATUS_1 : UDINT := UDINT#16#F086; (* < 61574 - PC1IS1 *)
    PGN_WIRELESS_CHARGER_SYSTEM_STATUS_1 : UDINT := UDINT#16#F087; (* < 61575 - WCSS1 *)
    PGN_WIRELESS_CHARGER_ALIGNMENT_QUALITY_STATUS : UDINT := UDINT#16#F088; (* < 61576 - WCAQS *)
    PGN_MOTOR_GENERATOR_1_INVERTER_CONTROL_STATUS_3 : UDINT := UDINT#16#F089; (* < 61577 - MG1IS3 *)
    PGN_MOTOR_GENERATOR_2_INVERTER_CONTROL_STATUS_3 : UDINT := UDINT#16#F08A; (* < 61578 - MG2IS3 *)
    PGN_MOTOR_GENERATOR_3_INVERTER_CONTROL_STATUS_3 : UDINT := UDINT#16#F08B; (* < 61579 - MG3IS3 *)
    PGN_MOTOR_GENERATOR_4_INVERTER_CONTROL_STATUS_3 : UDINT := UDINT#16#F08C; (* < 61580 - MG4IS3 *)
    PGN_MOTOR_GENERATOR_5_INVERTER_CONTROL_STATUS_3 : UDINT := UDINT#16#F08D; (* < 61581 - MG5IS3 *)
    PGN_MOTOR_GENERATOR_6_INVERTER_CONTROL_STATUS_3 : UDINT := UDINT#16#F08E; (* < 61582 - MG6IS3 *)
    PGN_HIGH_VOLTAGE_ENERGY_STORAGE_SYSTEM_DATA_1 : UDINT := UDINT#16#F090; (* < 61584 - HVESSD1 *)
    PGN_HIGH_VOLTAGE_ENERGY_STORAGE_SYSTEM_DATA_2 : UDINT := UDINT#16#F091; (* < 61585 - HVESSD2 *)
    PGN_HIGH_VOLTAGE_ENERGY_STORAGE_SYSTEM_DATA_3 : UDINT := UDINT#16#F092; (* < 61586 - HVESSD3 *)
    PGN_HIGH_VOLTAGE_ENERGY_STORAGE_SYSTEM_DATA_4 : UDINT := UDINT#16#F093; (* < 61587 - HVESSD4 *)
    PGN_HIGH_VOLTAGE_ENERGY_STORAGE_SYSTEM_DATA_5 : UDINT := UDINT#16#F094; (* < 61588 - HVESSD5 *)
    PGN_HIGH_VOLTAGE_ENERGY_STORAGE_SYSTEM_DATA_6 : UDINT := UDINT#16#F095; (* < 61589 - HVESSD6 *)
    PGN_HIGH_VOLTAGE_ENERGY_STORAGE_SYSTEM_STATUS_1 : UDINT := UDINT#16#F096; (* < 61590 - HVESSS1 *)
    PGN_MOTOR_GENERATOR_1_INVERTER_THERMAL_PERFORMANCE_STATUS : UDINT := UDINT#16#F097; (* < 61591 - MG1ITPS *)
    PGN_MOTOR_GENERATOR_2_INVERTER_THERMAL_PERFORMANCE_STATUS : UDINT := UDINT#16#F098; (* < 61592 - MG2ITPS *)
    PGN_MOTOR_GENERATOR_3_INVERTER_THERMAL_PERFORMANCE_STATUS : UDINT := UDINT#16#F099; (* < 61593 - MG3ITPS *)
    PGN_MOTOR_GENERATOR_4_INVERTER_THERMAL_PERFORMANCE_STATUS : UDINT := UDINT#16#F09A; (* < 61594 - MG4ITPS *)
    PGN_MOTOR_GENERATOR_5_INVERTER_THERMAL_PERFORMANCE_STATUS : UDINT := UDINT#16#F09B; (* < 61595 - MG5ITPS *)
    PGN_MOTOR_GENERATOR_6_INVERTER_THERMAL_PERFORMANCE_STATUS : UDINT := UDINT#16#F09C; (* < 61596 - MG6ITPS *)
    PGN_HIGH_VOLTAGE_ENERGY_STORAGE_SYSTEM_DATA_7 : UDINT := UDINT#16#F0A0; (* < 61600 - HVESSD7 *)
    PGN_DC_AC_ACCESSORY_INVERTER_1_STATUS_2 : UDINT := UDINT#16#F0C8; (* < 61640 - DCAC_AI1_S2 *)
    PGN_DC_AC_ACCESSORY_INVERTER_1_VOLTAGE : UDINT := UDINT#16#F0C9; (* < 61641 - DCAC_AI1_V *)
    PGN_DC_AC_ACCESSORY_INVERTER_1_FEEDBACK_2 : UDINT := UDINT#16#F0CA; (* < 61642 - DCAC_AI1_FDBK2 *)
    PGN_DC_AC_ACCESSORY_INVERTER_2_STATUS_2 : UDINT := UDINT#16#F0CB; (* < 61643 - DCAC_AI2_S2 *)
    PGN_DC_AC_ACCESSORY_INVERTER_2_VOLTAGE : UDINT := UDINT#16#F0CC; (* < 61644 - DCAC_AI2_V *)
    PGN_DC_AC_ACCESSORY_INVERTER_2_FEEDBACK_2 : UDINT := UDINT#16#F0CD; (* < 61645 - DCAC_AI2_FDBK2 *)
    PGN_ENGINE_TURBOCHARGER_CONTROL_4 : UDINT := UDINT#16#F0CE; (* < 61646 - ETCC4 *)
    PGN_ENGINE_TURBOCHARGER_WASTEGATE_ACTUATOR_AND_EXHAUST_BACK_PRESSURE_REGULATO_X : UDINT := UDINT#16#F0CF; (* < 61647 - ETWAI2 *)
    PGN_ENGINE_CYLINDER_COMBUSTION_REQUEST : UDINT := UDINT#16#F0D0; (* < 61648 - ECCR *)
    PGN_ENGINE_CYLINDER_HEAD_BYPASS_ACTUATOR_1 : UDINT := UDINT#16#F0D1; (* < 61649 - ECBA1 *)
    PGN_ENGINE_ELECTRONIC_CONTROLLER_18 : UDINT := UDINT#16#F0D2; (* < 61650 - EEC18 *)
    PGN_PREDICTIVE_CRUISE_CONTROL_1 : UDINT := UDINT#16#F0D3; (* < 61651 - PCC1 *)
    PGN_DC_AC_ACCESSORY_INVERTER_1_COMMAND : UDINT := UDINT#16#F0D6; (* < 61654 - DCAC_AI1_CMD *)
    PGN_DC_AC_ACCESSORY_INVERTER_1_FEEDBACK : UDINT := UDINT#16#F0D7; (* < 61655 - DCAC_AI1_FDBK *)
    PGN_DC_AC_ACCESSORY_INVERTER_2_COMMAND : UDINT := UDINT#16#F0DA; (* < 61658 - DCAC_AI2_CMD *)
    PGN_DC_AC_ACCESSORY_INVERTER_2_FEEDBACK : UDINT := UDINT#16#F0DB; (* < 61659 - DCAC_AI2_FDBK *)
    PGN_DC_AC_ACCESSORY_INVERTER_3_COMMAND : UDINT := UDINT#16#F0DE; (* < 61662 - DCAC_AI3_CMD *)
    PGN_DC_AC_ACCESSORY_INVERTER_3_FEEDBACK : UDINT := UDINT#16#F0DF; (* < 61663 - DCAC_AI3_FDBK *)
    PGN_DC_AC_ACCESSORY_INVERTER_4_COMMAND : UDINT := UDINT#16#F0E2; (* < 61666 - DCAC_AI4_CMD *)
    PGN_DC_AC_ACCESSORY_INVERTER_4_FEEDBACK : UDINT := UDINT#16#F0E3; (* < 61667 - DCAC_AI4_FDBK *)
    PGN_HEARTBEAT : UDINT := UDINT#16#F0E4; (* < 61668 - HRTBTM *)
    PGN_ENGINE_IGNITION_TIMING_OFFSET_1 : UDINT := UDINT#16#F0E5; (* < 61669 - ITO1 *)
    PGN_ENGINE_IGNITION_TIMING_OFFSET_2 : UDINT := UDINT#16#F0E6; (* < 61670 - ITO2 *)
    PGN_ENGINE_IGNITION_TIMING_OFFSET_3 : UDINT := UDINT#16#F0E7; (* < 61671 - ITO3 *)
    PGN_ENGINE_THROTTLE_FUEL_ACTUATOR_CONTROL_COMMAND_2 : UDINT := UDINT#16#F0E8; (* < 61672 - TFAC2 *)
    PGN_AFTERTREATMENT_1_INTAKE_GAS_3 : UDINT := UDINT#16#F0E9; (* < 61673 - AT1IG3 *)
    PGN_AFTERTREATMENT_1_OUTLET_GAS_3 : UDINT := UDINT#16#F0EA; (* < 61674 - AT1OG3 *)
    PGN_AFTERTREATMENT_2_INTAKE_GAS_3 : UDINT := UDINT#16#F0EB; (* < 61675 - AT2IG3 *)
    PGN_AFTERTREATMENT_2_OUTLET_GAS_3 : UDINT := UDINT#16#F0EC; (* < 61676 - AT2OG3 *)
    PGN_ENGINE_START_CONTROL : UDINT := UDINT#16#F0ED; (* < 61677 - ENGSC *)
    PGN_GENSET_REACTIVE_POWER_AND_SUPPORTING_FUNCTIONS : UDINT := UDINT#16#F0F4; (* < 61684 - GRPASF *)
    PGN_ENGINE_START_ARBITRATOR : UDINT := UDINT#16#F0F5; (* < 61685 - ENGSA *)
    PGN_ADVANCED_DRIVER_ASSISTANCE_SYSTEMS_INTERFACE_SPECIFICATION_1 : UDINT := UDINT#16#F0F6; (* < 61686 - ADASIS1 *)
    PGN_ADVANCED_DRIVER_ASSISTANCE_SYSTEMS_INTERFACE_SPECIFICATION_2 : UDINT := UDINT#16#F0F7; (* < 61687 - ADASIS2 *)
    PGN_ADVANCED_DRIVER_ASSISTANCE_SYSTEMS_INTERFACE_SPECIFICATION_3 : UDINT := UDINT#16#F0F8; (* < 61688 - ADASIS3 *)
    PGN_ENGINE_VALVE_CONTROLLER : UDINT := UDINT#16#F0F9; (* < 61689 - EVC *)
    PGN_ELECTRONIC_TRANSMISSION_CONTROLLER_13 : UDINT := UDINT#16#F0FA; (* < 61690 - ETC13 *)
    PGN_AFTERTREATMENT_1_SCR_DOSING_SYSTEM_REQUESTS_3 : UDINT := UDINT#16#F0FB; (* < 61691 - A1SCRDSR3 *)
    PGN_AFTERTREATMENT_2_SCR_DOSING_SYSTEM_REQUESTS_3 : UDINT := UDINT#16#F0FC; (* < 61692 - A2SCRDSR3 *)
    PGN_AFTERTREATMENT_1_SCR_DOSING_SYSTEM_INFORMATION_4 : UDINT := UDINT#16#F0FD; (* < 61693 - A1SCRDSI4 *)
    PGN_AFTERTREATMENT_2_SCR_DOSING_SYSTEM_INFORMATION_4 : UDINT := UDINT#16#F0FE; (* < 61694 - A2SCRDSI4 *)
    PGN_SECONDARY_OR_FRONT_HITCH_ROLL_AND_PITCH : UDINT := UDINT#16#F0FF; (* < 61695 - SHRP *)
    PGN_SECONDARY_OR_FRONT_HITCH_ROLL_AND_PITCH_COMMAND : UDINT := UDINT#16#F100; (* < 61696 - SHRPC *)
    PGN_PRIMARY_OR_REAR_HITCH_ROLL_AND_PITCH : UDINT := UDINT#16#F101; (* < 61697 - PHRP *)
    PGN_PRIMARY_OR_REAR_HITCH_ROLL_AND_PITCH_COMMAND : UDINT := UDINT#16#F102; (* < 61698 - PHRPC *)
    PGN_GENERATOR_TRIP_ENERGY : UDINT := UDINT#16#F103; (* < 61699 - GTRACE *)
    PGN_ENGINE_SPEED_SENSOR_INFORMATION_2 : UDINT := UDINT#16#F104; (* < 61700 - ESSI2 *)
    PGN_HYDRAULIC_PRESSURE_DISPLACEMENT : UDINT := UDINT#16#F105; (* < 61701 - HPD *)
    PGN_WELL_STIMULATION_PUMP_SYSTEM_1 : UDINT := UDINT#16#F106; (* < 61702 - WSP1 *)
    PGN_WELL_STIMULATION_PUMP_SYSTEM_2 : UDINT := UDINT#16#F107; (* < 61703 - WSP2 *)
    PGN_HIGH_VOLTAGE_ENERGY_STORAGE_SYSTEM_MODULE_STATUS_1 : UDINT := UDINT#16#F108; (* < 61704 - HVESSMS1 *)
    PGN_HIGH_VOLTAGE_ENERGY_STORAGE_SYSTEM_THERMAL_MANAGEMENT_SYSTEM_STATUS_1 : UDINT := UDINT#16#F109; (* < 61705 - HVESSTS1 *)
    PGN_HIGH_VOLTAGE_ENERGY_STORAGE_SYSTEM_DATA_8 : UDINT := UDINT#16#F10A; (* < 61706 - HVESSD8 *)
    PGN_HIGH_VOLTAGE_ENERGY_STORAGE_SYSTEM_DATA_9 : UDINT := UDINT#16#F10B; (* < 61707 - HVESSD9 *)
    PGN_HIGH_VOLTAGE_ENERGY_STORAGE_SYSTEM_DATA_10 : UDINT := UDINT#16#F10C; (* < 61708 - HVESSD10 *)
    PGN_FUEL_INFORMATION_6_GASEOUS : UDINT := UDINT#16#F10D; (* < 61709 - GFI6 *)
    PGN_DUMP_TRUCK_BODY_INFORMATION : UDINT := UDINT#16#F10E; (* < 61710 - DTBI1 *)
    PGN_ENGINE_OPERATING_INFORMATION_2 : UDINT := UDINT#16#F10F; (* < 61711 - EOI2 *)
    PGN_BRAKES_2 : UDINT := UDINT#16#F110; (* < 61712 - B2 *)
    PGN_GASEOUS_FUEL_PRESSURE_3 : UDINT := UDINT#16#F111; (* < 61713 - GFP3 *)
    PGN_DC_DC_CONVERTER_1_CONTROL : UDINT := UDINT#16#F112; (* < 61714 - DCDC1C *)
    PGN_DC_DC_CONVERTER_1_OPERATING_STATUS : UDINT := UDINT#16#F113; (* < 61715 - DCDC1OS *)
    PGN_DC_DC_CONVERTER_1_VOLTAGE_AND_CURRENT : UDINT := UDINT#16#F114; (* < 61716 - DCDC1VC *)
    PGN_DC_DC_CONVERTER_1_SLI_BATTERY_STATUS : UDINT := UDINT#16#F115; (* < 61717 - DCDC1SBS *)
    PGN_WELL_STIMULATION_PUMP_SYSTEM_3 : UDINT := UDINT#16#F116; (* < 61718 - WSP3 *)
    PGN_DC_DC_CONVERTER_1_STATUS_2 : UDINT := UDINT#16#F117; (* < 61719 - DCDC1S2 *)
    PGN_DC_DC_CONVERTER_2_CONTROL : UDINT := UDINT#16#F118; (* < 61720 - DCDC2C *)
    PGN_DC_DC_CONVERTER_2_OPERATING_STATUS : UDINT := UDINT#16#F119; (* < 61721 - DCDC2OS *)
    PGN_DC_DC_CONVERTER_2_VOLTAGE_AND_CURRENT : UDINT := UDINT#16#F11A; (* < 61722 - DCDC2VC *)
    PGN_DC_DC_CONVERTER_2_SLI_BATTERY_STATUS : UDINT := UDINT#16#F11B; (* < 61723 - DCDC2SBS *)
    PGN_DC_DC_CONVERTER_2_STATUS_2 : UDINT := UDINT#16#F11C; (* < 61724 - DCDC2S2 *)
    PGN_DC_DC_CONVERTER_3_CONTROL : UDINT := UDINT#16#F11D; (* < 61725 - DCDC3C *)
    PGN_DC_DC_CONVERTER_3_OPERATING_STATUS : UDINT := UDINT#16#F11E; (* < 61726 - DCDC3OS *)
    PGN_DC_DC_CONVERTER_3_VOLTAGE_AND_CURRENT : UDINT := UDINT#16#F11F; (* < 61727 - DCDC3VC *)
    PGN_DC_DC_CONVERTER_3_SLI_BATTERY_STATUS : UDINT := UDINT#16#F120; (* < 61728 - DCDC3SBS *)
    PGN_DC_DC_CONVERTER_3_STATUS_2 : UDINT := UDINT#16#F121; (* < 61729 - DCDC3S2 *)
    PGN_DC_DC_CONVERTER_4_CONTROL : UDINT := UDINT#16#F122; (* < 61730 - DCDC4C *)
    PGN_DC_DC_CONVERTER_4_OPERATING_STATUS : UDINT := UDINT#16#F123; (* < 61731 - DCDC4OS *)
    PGN_DC_DC_CONVERTER_4_VOLTAGE_AND_CURRENT : UDINT := UDINT#16#F124; (* < 61732 - DCDC4VC *)
    PGN_DC_DC_CONVERTER_4_SLI_BATTERY_STATUS : UDINT := UDINT#16#F125; (* < 61733 - DCDC4SBS *)
    PGN_DC_DC_CONVERTER_4_STATUS_2 : UDINT := UDINT#16#F126; (* < 61734 - DCDC4S2 *)
    PGN_SLOPE_SENSOR_INFORMATION_3 : UDINT := UDINT#16#F127; (* < 61735 - SSI3 *)
    PGN_DC_AC_ACCESSORY_INVERTER_3_STATUS_2 : UDINT := UDINT#16#F128; (* < 61736 - DCAC_AI3_S2 *)
    PGN_DC_AC_ACCESSORY_INVERTER_3_VOLTAGE : UDINT := UDINT#16#F129; (* < 61737 - DCAC_AI3_V *)
    PGN_DC_AC_ACCESSORY_INVERTER_3_FEEDBACK_2 : UDINT := UDINT#16#F12A; (* < 61738 - DCAC_AI3_FDBK2 *)
    PGN_DC_AC_ACCESSORY_INVERTER_4_STATUS_2 : UDINT := UDINT#16#F12B; (* < 61739 - DCAC_AI4_S2 *)
    PGN_DC_AC_ACCESSORY_INVERTER_4_VOLTAGE : UDINT := UDINT#16#F12C; (* < 61740 - DCAC_AI4_V *)
    PGN_DC_AC_ACCESSORY_INVERTER_4_FEEDBACK_2 : UDINT := UDINT#16#F12D; (* < 61741 - DCAC_AI4_FDBK2 *)
    PGN_DC_AC_ACCESSORY_INVERTER_5_COMMAND : UDINT := UDINT#16#F12E; (* < 61742 - DCAC_AI5_CMD *)
    PGN_DC_AC_ACCESSORY_INVERTER_5_FEEDBACK : UDINT := UDINT#16#F12F; (* < 61743 - DCAC_AI5_FDBK *)
    PGN_DC_AC_ACCESSORY_INVERTER_5_STATUS_2 : UDINT := UDINT#16#F130; (* < 61744 - DCAC_AI5_S2 *)
    PGN_DC_AC_ACCESSORY_INVERTER_5_VOLTAGE : UDINT := UDINT#16#F131; (* < 61745 - DCAC_AI5_V *)
    PGN_DC_AC_ACCESSORY_INVERTER_5_FEEDBACK_2 : UDINT := UDINT#16#F132; (* < 61746 - DCAC_AI5_FDBK2 *)
    PGN_ENGINE_PRE_CHAMBER_FUEL_VALVE_DURATION_COMMAND_1 : UDINT := UDINT#16#F133; (* < 61747 - EPCVDC1 *)
    PGN_ENGINE_PRE_CHAMBER_FUEL_VALVE_DURATION_COMMAND_2 : UDINT := UDINT#16#F134; (* < 61748 - EPCVDC2 *)
    PGN_ENGINE_PRE_CHAMBER_FUEL_VALVE_DURATION_COMMAND_3 : UDINT := UDINT#16#F135; (* < 61749 - EPCVDC3 *)
    PGN_ENGINE_PRE_CHAMBER_FUEL_VALVE_DURATION_COMMAND_4 : UDINT := UDINT#16#F136; (* < 61750 - EPCVDC4 *)
    PGN_ENGINE_PRE_CHAMBER_FUEL_VALVE_DURATION_COMMAND_5 : UDINT := UDINT#16#F137; (* < 61751 - EPCVDC5 *)
    PGN_ENGINE_PRE_CHAMBER_FUEL_VALVE_START_OF_ACTUATION_COMMAND_1 : UDINT := UDINT#16#F138; (* < 61752 - EPCSOAC1 *)
    PGN_ENGINE_PRE_CHAMBER_FUEL_VALVE_START_OF_ACTUATION_COMMAND_2 : UDINT := UDINT#16#F139; (* < 61753 - EPCSOAC2 *)
    PGN_ENGINE_PRE_CHAMBER_FUEL_VALVE_START_OF_ACTUATION_COMMAND_3 : UDINT := UDINT#16#F13A; (* < 61754 - EPCSOAC3 *)
    PGN_ENGINE_PRE_CHAMBER_FUEL_VALVE_START_OF_ACTUATION_COMMAND_4 : UDINT := UDINT#16#F13B; (* < 61755 - EPCSOAC4 *)
    PGN_ENGINE_PRE_CHAMBER_FUEL_VALVE_START_OF_ACTUATION_COMMAND_5 : UDINT := UDINT#16#F13C; (* < 61756 - EPCSOAC5 *)
    PGN_ACTIVE_STEERING_SYSTEM_CONTROLS_1 : UDINT := UDINT#16#F13D; (* < 61757 - ASSC1 *)
    PGN_SECONDARY_OR_FRONT_HITCH_YAW_COMMAND : UDINT := UDINT#16#F13E; (* < 61758 - FHYC *)
    PGN_PRIMARY_OR_REAR_HITCH_YAW_COMMAND : UDINT := UDINT#16#F13F; (* < 61759 - RHYC *)
    PGN_STATIONARY_INVERTER_AVERAGE_BASIC_AC_QUANTITIES : UDINT := UDINT#16#F140; (* < 61760 - SIAAC *)
    PGN_STATIONARY_INVERTER_TOTAL_AC_REACTIVE_POWER : UDINT := UDINT#16#F141; (* < 61761 - SITACR *)
    PGN_STATIONARY_INVERTER_TOTAL_AC_POWER : UDINT := UDINT#16#F142; (* < 61762 - SITACP *)
    PGN_STATIONARY_INVERTER_CONTROL : UDINT := UDINT#16#F143; (* < 61763 - SIC *)
    PGN_STATIONARY_INVERTER_TO_BUS_SYNC_CHECK_STATUS : UDINT := UDINT#16#F144; (* < 61764 - SIBSC *)
    PGN_ENGINE_CYLINDER_1_COMBUSTION_PRESSURES : UDINT := UDINT#16#F145; (* < 61765 - ECCP1 *)
    PGN_ENGINE_CYLINDER_2_COMBUSTION_PRESSURES : UDINT := UDINT#16#F146; (* < 61766 - ECCP2 *)
    PGN_ENGINE_CYLINDER_3_COMBUSTION_PRESSURES : UDINT := UDINT#16#F147; (* < 61767 - ECCP3 *)
    PGN_ENGINE_CYLINDER_4_COMBUSTION_PRESSURES : UDINT := UDINT#16#F148; (* < 61768 - ECCP4 *)
    PGN_ENGINE_CYLINDER_5_COMBUSTION_PRESSURES : UDINT := UDINT#16#F149; (* < 61769 - ECCP5 *)
    PGN_ENGINE_CYLINDER_6_COMBUSTION_PRESSURES : UDINT := UDINT#16#F14A; (* < 61770 - ECCP6 *)
    PGN_ENGINE_CYLINDER_7_COMBUSTION_PRESSURES : UDINT := UDINT#16#F14B; (* < 61771 - ECCP7 *)
    PGN_ENGINE_CYLINDER_8_COMBUSTION_PRESSURES : UDINT := UDINT#16#F14C; (* < 61772 - ECCP8 *)
    PGN_ENGINE_CYLINDER_9_COMBUSTION_PRESSURES : UDINT := UDINT#16#F14D; (* < 61773 - ECCP9 *)
    PGN_ENGINE_CYLINDER_10_COMBUSTION_PRESSURES : UDINT := UDINT#16#F14E; (* < 61774 - ECCP10 *)
    PGN_ENGINE_CYLINDER_11_COMBUSTION_PRESSURES : UDINT := UDINT#16#F14F; (* < 61775 - ECCP11 *)
    PGN_ENGINE_CYLINDER_12_COMBUSTION_PRESSURES : UDINT := UDINT#16#F150; (* < 61776 - ECCP12 *)
    PGN_ENGINE_CYLINDER_13_COMBUSTION_PRESSURES : UDINT := UDINT#16#F151; (* < 61777 - ECCP13 *)
    PGN_ENGINE_CYLINDER_14_COMBUSTION_PRESSURES : UDINT := UDINT#16#F152; (* < 61778 - ECCP14 *)
    PGN_ENGINE_CYLINDER_15_COMBUSTION_PRESSURES : UDINT := UDINT#16#F153; (* < 61779 - ECCP15 *)
    PGN_ENGINE_CYLINDER_16_COMBUSTION_PRESSURES : UDINT := UDINT#16#F154; (* < 61780 - ECCP16 *)
    PGN_ENGINE_CYLINDER_17_COMBUSTION_PRESSURES : UDINT := UDINT#16#F155; (* < 61781 - ECCP17 *)
    PGN_ENGINE_CYLINDER_18_COMBUSTION_PRESSURES : UDINT := UDINT#16#F156; (* < 61782 - ECCP18 *)
    PGN_ENGINE_CYLINDER_19_COMBUSTION_PRESSURES : UDINT := UDINT#16#F157; (* < 61783 - ECCP19 *)
    PGN_ENGINE_CYLINDER_20_COMBUSTION_PRESSURES : UDINT := UDINT#16#F158; (* < 61784 - ECCP20 *)
    PGN_ENGINE_CYLINDER_1_COMBUSTION_TIMING : UDINT := UDINT#16#F159; (* < 61785 - ECCT1 *)
    PGN_ENGINE_CYLINDER_2_COMBUSTION_TIMING : UDINT := UDINT#16#F15A; (* < 61786 - ECCT2 *)
    PGN_ENGINE_CYLINDER_3_COMBUSTION_TIMING : UDINT := UDINT#16#F15B; (* < 61787 - ECCT3 *)
    PGN_ENGINE_CYLINDER_4_COMBUSTION_TIMING : UDINT := UDINT#16#F15C; (* < 61788 - ECCT4 *)
    PGN_ENGINE_CYLINDER_5_COMBUSTION_TIMING : UDINT := UDINT#16#F15D; (* < 61789 - ECCT5 *)
    PGN_ENGINE_CYLINDER_6_COMBUSTION_TIMING : UDINT := UDINT#16#F15E; (* < 61790 - ECCT6 *)
    PGN_ENGINE_CYLINDER_7_COMBUSTION_TIMING : UDINT := UDINT#16#F15F; (* < 61791 - ECCT7 *)
    PGN_ENGINE_CYLINDER_8_COMBUSTION_TIMING : UDINT := UDINT#16#F160; (* < 61792 - ECCT8 *)
    PGN_ENGINE_CYLINDER_9_COMBUSTION_TIMING : UDINT := UDINT#16#F161; (* < 61793 - ECCT9 *)
    PGN_ENGINE_CYLINDER_10_COMBUSTION_TIMING : UDINT := UDINT#16#F162; (* < 61794 - ECCT10 *)
    PGN_ENGINE_CYLINDER_11_COMBUSTION_TIMING : UDINT := UDINT#16#F163; (* < 61795 - ECCT11 *)
    PGN_ENGINE_CYLINDER_12_COMBUSTION_TIMING : UDINT := UDINT#16#F164; (* < 61796 - ECCT12 *)
    PGN_ENGINE_CYLINDER_13_COMBUSTION_TIMING : UDINT := UDINT#16#F165; (* < 61797 - ECCT13 *)
    PGN_ENGINE_CYLINDER_14_COMBUSTION_TIMING : UDINT := UDINT#16#F166; (* < 61798 - ECCT14 *)
    PGN_ENGINE_CYLINDER_15_COMBUSTION_TIMING : UDINT := UDINT#16#F167; (* < 61799 - ECCT15 *)
    PGN_ENGINE_CYLINDER_16_COMBUSTION_TIMING : UDINT := UDINT#16#F168; (* < 61800 - ECCT16 *)
    PGN_ENGINE_CYLINDER_17_COMBUSTION_TIMING : UDINT := UDINT#16#F169; (* < 61801 - ECCT17 *)
    PGN_ENGINE_CYLINDER_18_COMBUSTION_TIMING : UDINT := UDINT#16#F16A; (* < 61802 - ECCT18 *)
    PGN_ENGINE_CYLINDER_19_COMBUSTION_TIMING : UDINT := UDINT#16#F16B; (* < 61803 - ECCT19 *)
    PGN_ENGINE_CYLINDER_20_COMBUSTION_TIMING : UDINT := UDINT#16#F16C; (* < 61804 - ECCT20 *)
    PGN_ENGINE_CYLINDER_1_COMBUSTION_METRICS : UDINT := UDINT#16#F16D; (* < 61805 - EECM1 *)
    PGN_ENGINE_CYLINDER_2_COMBUSTION_METRICS : UDINT := UDINT#16#F16E; (* < 61806 - EECM2 *)
    PGN_ENGINE_CYLINDER_3_COMBUSTION_METRICS : UDINT := UDINT#16#F16F; (* < 61807 - EECM3 *)
    PGN_ENGINE_CYLINDER_4_COMBUSTION_METRICS : UDINT := UDINT#16#F170; (* < 61808 - EECM4 *)
    PGN_ENGINE_CYLINDER_5_COMBUSTION_METRICS : UDINT := UDINT#16#F171; (* < 61809 - EECM5 *)
    PGN_ENGINE_CYLINDER_6_COMBUSTION_METRICS : UDINT := UDINT#16#F172; (* < 61810 - EECM6 *)
    PGN_ENGINE_CYLINDER_7_COMBUSTION_METRICS : UDINT := UDINT#16#F173; (* < 61811 - EECM7 *)
    PGN_ENGINE_CYLINDER_8_COMBUSTION_METRICS : UDINT := UDINT#16#F174; (* < 61812 - EECM8 *)
    PGN_ENGINE_CYLINDER_9_COMBUSTION_METRICS : UDINT := UDINT#16#F175; (* < 61813 - EECM9 *)
    PGN_ENGINE_CYLINDER_10_COMBUSTION_METRICS : UDINT := UDINT#16#F176; (* < 61814 - EECM10 *)
    PGN_ENGINE_CYLINDER_11_COMBUSTION_METRICS : UDINT := UDINT#16#F177; (* < 61815 - EECM11 *)
    PGN_ENGINE_CYLINDER_12_COMBUSTION_METRICS : UDINT := UDINT#16#F178; (* < 61816 - EECM12 *)
    PGN_ENGINE_CYLINDER_13_COMBUSTION_METRICS : UDINT := UDINT#16#F179; (* < 61817 - EECM13 *)
    PGN_ENGINE_CYLINDER_14_COMBUSTION_METRICS : UDINT := UDINT#16#F17A; (* < 61818 - EECM14 *)
    PGN_ENGINE_CYLINDER_15_COMBUSTION_METRICS : UDINT := UDINT#16#F17B; (* < 61819 - EECM15 *)
    PGN_ENGINE_CYLINDER_16_COMBUSTION_METRICS : UDINT := UDINT#16#F17C; (* < 61820 - EECM16 *)
    PGN_ENGINE_CYLINDER_17_COMBUSTION_METRICS : UDINT := UDINT#16#F17D; (* < 61821 - EECM17 *)
    PGN_ENGINE_CYLINDER_18_COMBUSTION_METRICS : UDINT := UDINT#16#F17E; (* < 61822 - EECM18 *)
    PGN_ENGINE_CYLINDER_19_COMBUSTION_METRICS : UDINT := UDINT#16#F17F; (* < 61823 - EECM19 *)
    PGN_ENGINE_CYLINDER_20_COMBUSTION_METRICS : UDINT := UDINT#16#F180; (* < 61824 - EECM20 *)
    PGN_MOTOR_GENERATOR_1_INVERTER_MODE_FEEDBACK_1 : UDINT := UDINT#16#F181; (* < 61825 - MG1IMF1 *)
    PGN_MOTOR_GENERATOR_1_INVERTER_LIMITS_ACTIVE_POWER : UDINT := UDINT#16#F182; (* < 61826 - MG1ILAP *)
    PGN_MOTOR_GENERATOR_1_INVERTER_LIMITS_ACTIVE_MECHANICAL : UDINT := UDINT#16#F183; (* < 61827 - MG1ILAM *)
    PGN_MOTOR_GENERATOR_1_INVERTER_LIMITS_ACTIVE_DC_SIDE : UDINT := UDINT#16#F184; (* < 61828 - MG1ILADC *)
    PGN_MOTOR_GENERATOR_1_INVERTER_LOW_VOLTAGE : UDINT := UDINT#16#F185; (* < 61829 - MG1ILV *)
    PGN_MOTOR_GENERATOR_2_INVERTER_MODE_FEEDBACK_1 : UDINT := UDINT#16#F186; (* < 61830 - MG2IMF1 *)
    PGN_MOTOR_GENERATOR_2_INVERTER_LIMITS_ACTIVE_POWER : UDINT := UDINT#16#F187; (* < 61831 - MG2ILAP *)
    PGN_MOTOR_GENERATOR_2_INVERTER_LIMITS_ACTIVE_MECHANICAL : UDINT := UDINT#16#F188; (* < 61832 - MG2ILAM *)
    PGN_MOTOR_GENERATOR_2_INVERTER_LIMITS_ACTIVE_DC_SIDE : UDINT := UDINT#16#F189; (* < 61833 - MG2ILADC *)
    PGN_MOTOR_GENERATOR_2_INVERTER_LOW_VOLTAGE : UDINT := UDINT#16#F18A; (* < 61834 - MG2ILV *)
    PGN_MOTOR_GENERATOR_1_INVERTER_STATUS_2 : UDINT := UDINT#16#F18B; (* < 61835 - MG1IS2 *)
    PGN_MOTOR_GENERATOR_1_INVERTER_RATE_LIMITS_ACTIVE_1 : UDINT := UDINT#16#F18C; (* < 61836 - MG1IRLA1 *)
    PGN_MOTOR_GENERATOR_2_INVERTER_STATUS_2 : UDINT := UDINT#16#F18D; (* < 61837 - MG2IS2 *)
    PGN_MOTOR_GENERATOR_2_INVERTER_RATE_LIMITS_ACTIVE_1 : UDINT := UDINT#16#F18E; (* < 61838 - MG2IRLA1 *)
    PGN_IMPOSTOR_PG_ALERT : UDINT := UDINT#16#F18F; (* < 61839 - IPGA *)
    PGN_HIGH_VOLTAGE_ENERGY_STORAGE_PACK_1_STATUS_2 : UDINT := UDINT#16#F190; (* < 61840 - HVESP1S2 *)
    PGN_HIGH_VOLTAGE_ENERGY_STORAGE_PACK_1_DATA_1 : UDINT := UDINT#16#F191; (* < 61841 - HVESP1D1 *)
    PGN_HIGH_VOLTAGE_ENERGY_STORAGE_PACK_1_DATA_2 : UDINT := UDINT#16#F192; (* < 61842 - HVESP1D2 *)
    PGN_HIGH_VOLTAGE_ENERGY_STORAGE_PACK_1_DATA_3 : UDINT := UDINT#16#F193; (* < 61843 - HVESP1D3 *)
    PGN_HIGH_VOLTAGE_ENERGY_STORAGE_PACK_1_DATA_4 : UDINT := UDINT#16#F194; (* < 61844 - HVESP1D4 *)
    PGN_HIGH_VOLTAGE_ENERGY_STORAGE_PACK_1_DATA_5 : UDINT := UDINT#16#F195; (* < 61845 - HVESP1D5 *)
    PGN_HIGH_VOLTAGE_ENERGY_STORAGE_PACK_1_DATA_6 : UDINT := UDINT#16#F196; (* < 61846 - HVESP1D6 *)
    PGN_HIGH_VOLTAGE_ENERGY_STORAGE_PACK_1_STATUS_1 : UDINT := UDINT#16#F197; (* < 61847 - HVESP1S1 *)
    PGN_HIGH_VOLTAGE_ENERGY_STORAGE_PACK_1_DATA_7 : UDINT := UDINT#16#F198; (* < 61848 - HVESP1D7 *)
    PGN_HIGH_VOLTAGE_ENERGY_STORAGE_PACK_1_MODULE_STATUS_1 : UDINT := UDINT#16#F199; (* < 61849 - HVESP1MS1 *)
    PGN_HIGH_VOLTAGE_ENERGY_STORAGE_PACK_1_THERMAL_MANAGEMENT_SYSTEM_STATUS_1 : UDINT := UDINT#16#F19A; (* < 61850 - HVESP1TS1 *)
    PGN_HIGH_VOLTAGE_ENERGY_STORAGE_PACK_1_DATA_8 : UDINT := UDINT#16#F19B; (* < 61851 - HVESP1D8 *)
    PGN_HIGH_VOLTAGE_ENERGY_STORAGE_PACK_1_DATA_9 : UDINT := UDINT#16#F19C; (* < 61852 - HVESP1D9 *)
    PGN_HIGH_VOLTAGE_ENERGY_STORAGE_PACK_1_DATA_10 : UDINT := UDINT#16#F19D; (* < 61853 - HVESP1D10 *)
    PGN_HIGH_VOLTAGE_ENERGY_STORAGE_PACK_1_DATA_11 : UDINT := UDINT#16#F19E; (* < 61854 - HVESP1D11 *)
    PGN_HIGH_VOLTAGE_ENERGY_STORAGE_PACK_2_STATUS_2 : UDINT := UDINT#16#F19F; (* < 61855 - HVESP2S2 *)
    PGN_HIGH_VOLTAGE_ENERGY_STORAGE_PACK_2_DATA_1 : UDINT := UDINT#16#F1A0; (* < 61856 - HVESP2D1 *)
    PGN_HIGH_VOLTAGE_ENERGY_STORAGE_PACK_2_DATA_2 : UDINT := UDINT#16#F1A1; (* < 61857 - HVESP2D2 *)
    PGN_HIGH_VOLTAGE_ENERGY_STORAGE_PACK_2_DATA_3 : UDINT := UDINT#16#F1A2; (* < 61858 - HVESP2D3 *)
    PGN_HIGH_VOLTAGE_ENERGY_STORAGE_PACK_2_DATA_4 : UDINT := UDINT#16#F1A3; (* < 61859 - HVESP2D4 *)
    PGN_HIGH_VOLTAGE_ENERGY_STORAGE_PACK_2_DATA_5 : UDINT := UDINT#16#F1A4; (* < 61860 - HVESP2D5 *)
    PGN_HIGH_VOLTAGE_ENERGY_STORAGE_PACK_2_DATA_6 : UDINT := UDINT#16#F1A5; (* < 61861 - HVESP2D6 *)
    PGN_HIGH_VOLTAGE_ENERGY_STORAGE_PACK_2_STATUS_1 : UDINT := UDINT#16#F1A6; (* < 61862 - HVESP2S1 *)
    PGN_HIGH_VOLTAGE_ENERGY_STORAGE_PACK_2_DATA_7 : UDINT := UDINT#16#F1A7; (* < 61863 - HVESP2D7 *)
    PGN_HIGH_VOLTAGE_ENERGY_STORAGE_PACK_2_MODULE_STATUS_1 : UDINT := UDINT#16#F1A8; (* < 61864 - HVESP2MS1 *)
    PGN_HIGH_VOLTAGE_ENERGY_STORAGE_PACK_2_THERMAL_MANAGEMENT_SYSTEM_STATUS_1 : UDINT := UDINT#16#F1A9; (* < 61865 - HVESP2TS1 *)
    PGN_HIGH_VOLTAGE_ENERGY_STORAGE_PACK_2_DATA_8 : UDINT := UDINT#16#F1AA; (* < 61866 - HVESP2D8 *)
    PGN_HIGH_VOLTAGE_ENERGY_STORAGE_PACK_2_DATA_9 : UDINT := UDINT#16#F1AB; (* < 61867 - HVESP2D9 *)
    PGN_HIGH_VOLTAGE_ENERGY_STORAGE_PACK_2_DATA_10 : UDINT := UDINT#16#F1AC; (* < 61868 - HVESP2D10 *)
    PGN_HIGH_VOLTAGE_ENERGY_STORAGE_PACK_2_DATA_11 : UDINT := UDINT#16#F1AD; (* < 61869 - HVESP2D11 *)
    PGN_HIGH_VOLTAGE_ENERGY_STORAGE_PACK_3_STATUS_2 : UDINT := UDINT#16#F1AE; (* < 61870 - HVESP3S2 *)
    PGN_HIGH_VOLTAGE_ENERGY_STORAGE_PACK_3_DATA_1 : UDINT := UDINT#16#F1AF; (* < 61871 - HVESP3D1 *)
    PGN_HIGH_VOLTAGE_ENERGY_STORAGE_PACK_3_DATA_2 : UDINT := UDINT#16#F1B0; (* < 61872 - HVESP3D2 *)
    PGN_HIGH_VOLTAGE_ENERGY_STORAGE_PACK_3_DATA_3 : UDINT := UDINT#16#F1B1; (* < 61873 - HVESP3D3 *)
    PGN_HIGH_VOLTAGE_ENERGY_STORAGE_PACK_3_DATA_4 : UDINT := UDINT#16#F1B2; (* < 61874 - HVESP3D4 *)
    PGN_HIGH_VOLTAGE_ENERGY_STORAGE_PACK_3_DATA_5 : UDINT := UDINT#16#F1B3; (* < 61875 - HVESP3D5 *)
    PGN_HIGH_VOLTAGE_ENERGY_STORAGE_PACK_3_DATA_6 : UDINT := UDINT#16#F1B4; (* < 61876 - HVESP3D6 *)
    PGN_HIGH_VOLTAGE_ENERGY_STORAGE_PACK_3_STATUS_1 : UDINT := UDINT#16#F1B5; (* < 61877 - HVESP3S1 *)
    PGN_HIGH_VOLTAGE_ENERGY_STORAGE_PACK_3_DATA_7 : UDINT := UDINT#16#F1B6; (* < 61878 - HVESP3D7 *)
    PGN_HIGH_VOLTAGE_ENERGY_STORAGE_PACK_3_MODULE_STATUS_1 : UDINT := UDINT#16#F1B7; (* < 61879 - HVESP3MS1 *)
    PGN_HIGH_VOLTAGE_ENERGY_STORAGE_PACK_3_THERMAL_MANAGEMENT_SYSTEM_STATUS_1 : UDINT := UDINT#16#F1B8; (* < 61880 - HVESP3TS1 *)
    PGN_HIGH_VOLTAGE_ENERGY_STORAGE_PACK_3_DATA_8 : UDINT := UDINT#16#F1B9; (* < 61881 - HVESP3D8 *)
    PGN_HIGH_VOLTAGE_ENERGY_STORAGE_PACK_3_DATA_9 : UDINT := UDINT#16#F1BA; (* < 61882 - HVESP3D9 *)
    PGN_HIGH_VOLTAGE_ENERGY_STORAGE_PACK_3_DATA_10 : UDINT := UDINT#16#F1BB; (* < 61883 - HVESP3D10 *)
    PGN_HIGH_VOLTAGE_ENERGY_STORAGE_PACK_3_DATA_11 : UDINT := UDINT#16#F1BC; (* < 61884 - HVESP3D11 *)
    PGN_HIGH_VOLTAGE_ENERGY_STORAGE_PACK_4_STATUS_2 : UDINT := UDINT#16#F1BD; (* < 61885 - HVESP4S2 *)
    PGN_HIGH_VOLTAGE_ENERGY_STORAGE_PACK_4_DATA_1 : UDINT := UDINT#16#F1BE; (* < 61886 - HVESP4D1 *)
    PGN_HIGH_VOLTAGE_ENERGY_STORAGE_PACK_4_DATA_2 : UDINT := UDINT#16#F1BF; (* < 61887 - HVESP4D2 *)
    PGN_HIGH_VOLTAGE_ENERGY_STORAGE_PACK_4_DATA_3 : UDINT := UDINT#16#F1C0; (* < 61888 - HVESP4D3 *)
    PGN_HIGH_VOLTAGE_ENERGY_STORAGE_PACK_4_DATA_4 : UDINT := UDINT#16#F1C1; (* < 61889 - HVESP4D4 *)
    PGN_HIGH_VOLTAGE_ENERGY_STORAGE_PACK_4_DATA_5 : UDINT := UDINT#16#F1C2; (* < 61890 - HVESP4D5 *)
    PGN_HIGH_VOLTAGE_ENERGY_STORAGE_PACK_4_DATA_6 : UDINT := UDINT#16#F1C3; (* < 61891 - HVESP4D6 *)
    PGN_HIGH_VOLTAGE_ENERGY_STORAGE_PACK_4_STATUS_1 : UDINT := UDINT#16#F1C4; (* < 61892 - HVESP4S1 *)
    PGN_HIGH_VOLTAGE_ENERGY_STORAGE_PACK_4_DATA_7 : UDINT := UDINT#16#F1C5; (* < 61893 - HVESP4D7 *)
    PGN_HIGH_VOLTAGE_ENERGY_STORAGE_PACK_4_MODULE_STATUS_1 : UDINT := UDINT#16#F1C6; (* < 61894 - HVESP4MS1 *)
    PGN_HIGH_VOLTAGE_ENERGY_STORAGE_PACK_4_THERMAL_MANAGEMENT_SYSTEM_STATUS_1 : UDINT := UDINT#16#F1C7; (* < 61895 - HVESP4TS1 *)
    PGN_HIGH_VOLTAGE_ENERGY_STORAGE_PACK_4_DATA_8 : UDINT := UDINT#16#F1C8; (* < 61896 - HVESP4D8 *)
    PGN_HIGH_VOLTAGE_ENERGY_STORAGE_PACK_4_DATA_9 : UDINT := UDINT#16#F1C9; (* < 61897 - HVESP4D9 *)
    PGN_HIGH_VOLTAGE_ENERGY_STORAGE_PACK_4_DATA_10 : UDINT := UDINT#16#F1CA; (* < 61898 - HVESP4D10 *)
    PGN_HIGH_VOLTAGE_ENERGY_STORAGE_PACK_4_DATA_11 : UDINT := UDINT#16#F1CB; (* < 61899 - HVESP4D11 *)
    PGN_HIGH_VOLTAGE_ENERGY_STORAGE_PACK_5_STATUS_2 : UDINT := UDINT#16#F1CC; (* < 61900 - HVESP5S2 *)
    PGN_HIGH_VOLTAGE_ENERGY_STORAGE_PACK_5_DATA_1 : UDINT := UDINT#16#F1CD; (* < 61901 - HVESP5D1 *)
    PGN_HIGH_VOLTAGE_ENERGY_STORAGE_PACK_5_DATA_2 : UDINT := UDINT#16#F1CE; (* < 61902 - HVESP5D2 *)
    PGN_HIGH_VOLTAGE_ENERGY_STORAGE_PACK_5_DATA_3 : UDINT := UDINT#16#F1CF; (* < 61903 - HVESP5D3 *)
    PGN_HIGH_VOLTAGE_ENERGY_STORAGE_PACK_5_DATA_4 : UDINT := UDINT#16#F1D0; (* < 61904 - HVESP5D4 *)
    PGN_HIGH_VOLTAGE_ENERGY_STORAGE_PACK_5_DATA_5 : UDINT := UDINT#16#F1D1; (* < 61905 - HVESP5D5 *)
    PGN_HIGH_VOLTAGE_ENERGY_STORAGE_PACK_5_DATA_6 : UDINT := UDINT#16#F1D2; (* < 61906 - HVESP5D6 *)
    PGN_HIGH_VOLTAGE_ENERGY_STORAGE_PACK_5_STATUS_1 : UDINT := UDINT#16#F1D3; (* < 61907 - HVESP5S1 *)
    PGN_HIGH_VOLTAGE_ENERGY_STORAGE_PACK_5_DATA_7 : UDINT := UDINT#16#F1D4; (* < 61908 - HVESP5D7 *)
    PGN_HIGH_VOLTAGE_ENERGY_STORAGE_PACK_5_MODULE_STATUS_1 : UDINT := UDINT#16#F1D5; (* < 61909 - HVESP5MS1 *)
    PGN_HIGH_VOLTAGE_ENERGY_STORAGE_PACK_5_THERMAL_MANAGEMENT_SYSTEM_STATUS_1 : UDINT := UDINT#16#F1D6; (* < 61910 - HVESP5TS1 *)
    PGN_HIGH_VOLTAGE_ENERGY_STORAGE_PACK_5_DATA_8 : UDINT := UDINT#16#F1D7; (* < 61911 - HVESP5D8 *)
    PGN_HIGH_VOLTAGE_ENERGY_STORAGE_PACK_5_DATA_9 : UDINT := UDINT#16#F1D8; (* < 61912 - HVESP5D9 *)
    PGN_HIGH_VOLTAGE_ENERGY_STORAGE_PACK_5_DATA_10 : UDINT := UDINT#16#F1D9; (* < 61913 - HVESP5D10 *)
    PGN_HIGH_VOLTAGE_ENERGY_STORAGE_PACK_5_DATA_11 : UDINT := UDINT#16#F1DA; (* < 61914 - HVESP5D11 *)
    PGN_HIGH_VOLTAGE_ENERGY_STORAGE_PACK_6_STATUS_2 : UDINT := UDINT#16#F1DB; (* < 61915 - HVESP6S2 *)
    PGN_HIGH_VOLTAGE_ENERGY_STORAGE_PACK_6_DATA_1 : UDINT := UDINT#16#F1DC; (* < 61916 - HVESP6D1 *)
    PGN_HIGH_VOLTAGE_ENERGY_STORAGE_PACK_6_DATA_2 : UDINT := UDINT#16#F1DD; (* < 61917 - HVESP6D2 *)
    PGN_HIGH_VOLTAGE_ENERGY_STORAGE_PACK_6_DATA_3 : UDINT := UDINT#16#F1DE; (* < 61918 - HVESP6D3 *)
    PGN_HIGH_VOLTAGE_ENERGY_STORAGE_PACK_6_DATA_4 : UDINT := UDINT#16#F1DF; (* < 61919 - HVESP6D4 *)
    PGN_HIGH_VOLTAGE_ENERGY_STORAGE_PACK_6_DATA_5 : UDINT := UDINT#16#F1E0; (* < 61920 - HVESP6D5 *)
    PGN_HIGH_VOLTAGE_ENERGY_STORAGE_PACK_6_DATA_6 : UDINT := UDINT#16#F1E1; (* < 61921 - HVESP6D6 *)
    PGN_HIGH_VOLTAGE_ENERGY_STORAGE_PACK_6_STATUS_1 : UDINT := UDINT#16#F1E2; (* < 61922 - HVESP6S1 *)
    PGN_HIGH_VOLTAGE_ENERGY_STORAGE_PACK_6_DATA_7 : UDINT := UDINT#16#F1E3; (* < 61923 - HVESP6D7 *)
    PGN_HIGH_VOLTAGE_ENERGY_STORAGE_PACK_6_MODULE_STATUS_1 : UDINT := UDINT#16#F1E4; (* < 61924 - HVESP6MS1 *)
    PGN_HIGH_VOLTAGE_ENERGY_STORAGE_PACK_6_THERMAL_MANAGEMENT_SYSTEM_STATUS_1 : UDINT := UDINT#16#F1E5; (* < 61925 - HVESP6TS1 *)
    PGN_HIGH_VOLTAGE_ENERGY_STORAGE_PACK_6_DATA_8 : UDINT := UDINT#16#F1E6; (* < 61926 - HVESP6D8 *)
    PGN_HIGH_VOLTAGE_ENERGY_STORAGE_PACK_6_DATA_9 : UDINT := UDINT#16#F1E7; (* < 61927 - HVESP6D9 *)
    PGN_HIGH_VOLTAGE_ENERGY_STORAGE_PACK_6_DATA_10 : UDINT := UDINT#16#F1E8; (* < 61928 - HVESP6D10 *)
    PGN_HIGH_VOLTAGE_ENERGY_STORAGE_PACK_6_DATA_11 : UDINT := UDINT#16#F1E9; (* < 61929 - HVESP6D11 *)
    PGN_MOTOR_GENERATOR_3_INVERTER_MODE_FEEDBACK_1 : UDINT := UDINT#16#F1EA; (* < 61930 - MG3IMF1 *)
    PGN_MOTOR_GENERATOR_3_INVERTER_LIMITS_ACTIVE_POWER : UDINT := UDINT#16#F1EB; (* < 61931 - MG3ILAP *)
    PGN_MOTOR_GENERATOR_3_INVERTER_LIMITS_ACTIVE_MECHANICAL : UDINT := UDINT#16#F1EC; (* < 61932 - MG3ILAM *)
    PGN_MOTOR_GENERATOR_3_INVERTER_LIMITS_ACTIVE_DC_SIDE : UDINT := UDINT#16#F1ED; (* < 61933 - MG3ILADC *)
    PGN_MOTOR_GENERATOR_3_INVERTER_LOW_VOLTAGE : UDINT := UDINT#16#F1EE; (* < 61934 - MG3ILV *)
    PGN_MOTOR_GENERATOR_3_INVERTER_STATUS_2 : UDINT := UDINT#16#F1EF; (* < 61935 - MG3IS2 *)
    PGN_MOTOR_GENERATOR_3_INVERTER_RATE_LIMITS_ACTIVE_1 : UDINT := UDINT#16#F1F0; (* < 61936 - MG3IRLA1 *)
    PGN_MOTOR_GENERATOR_4_INVERTER_MODE_FEEDBACK_1 : UDINT := UDINT#16#F1F1; (* < 61937 - MG4IMF1 *)
    PGN_MOTOR_GENERATOR_4_INVERTER_LIMITS_ACTIVE_POWER : UDINT := UDINT#16#F1F2; (* < 61938 - MG4ILAP *)
    PGN_MOTOR_GENERATOR_4_INVERTER_LIMITS_ACTIVE_MECHANICAL : UDINT := UDINT#16#F1F3; (* < 61939 - MG4ILAM *)
    PGN_MOTOR_GENERATOR_4_INVERTER_LIMITS_ACTIVE_DC_SIDE : UDINT := UDINT#16#F1F4; (* < 61940 - MG4ILADC *)
    PGN_MOTOR_GENERATOR_4_INVERTER_LOW_VOLTAGE : UDINT := UDINT#16#F1F5; (* < 61941 - MG4ILV *)
    PGN_MOTOR_GENERATOR_4_INVERTER_STATUS_2 : UDINT := UDINT#16#F1F6; (* < 61942 - MG4IS2 *)
    PGN_MOTOR_GENERATOR_4_INVERTER_RATE_LIMITS_ACTIVE_1 : UDINT := UDINT#16#F1F7; (* < 61943 - MG4IRLA1 *)
    PGN_MOTOR_GENERATOR_5_INVERTER_MODE_FEEDBACK_1 : UDINT := UDINT#16#F1F8; (* < 61944 - MG5IMF1 *)
    PGN_MOTOR_GENERATOR_5_INVERTER_LIMITS_ACTIVE_POWER : UDINT := UDINT#16#F1F9; (* < 61945 - MG5ILAP *)
    PGN_MOTOR_GENERATOR_5_INVERTER_LIMITS_ACTIVE_MECHANICAL : UDINT := UDINT#16#F1FA; (* < 61946 - MG5ILAM *)
    PGN_MOTOR_GENERATOR_5_INVERTER_LIMITS_ACTIVE_DC_SIDE : UDINT := UDINT#16#F1FB; (* < 61947 - MG5ILADC *)
    PGN_MOTOR_GENERATOR_5_INVERTER_LOW_VOLTAGE : UDINT := UDINT#16#F1FC; (* < 61948 - MG5ILV *)
    PGN_MOTOR_GENERATOR_5_INVERTER_STATUS_2 : UDINT := UDINT#16#F1FD; (* < 61949 - MG5IS2 *)
    PGN_MOTOR_GENERATOR_5_INVERTER_RATE_LIMITS_ACTIVE_1 : UDINT := UDINT#16#F1FE; (* < 61950 - MG5IRLA1 *)
    PGN_MOTOR_GENERATOR_6_INVERTER_MODE_FEEDBACK_1 : UDINT := UDINT#16#F1FF; (* < 61951 - MG6IMF1 *)
    PGN_MOTOR_GENERATOR_6_INVERTER_LIMITS_ACTIVE_POWER : UDINT := UDINT#16#F200; (* < 61952 - MG6ILAP *)
    PGN_MOTOR_GENERATOR_6_INVERTER_LIMITS_ACTIVE_MECHANICAL : UDINT := UDINT#16#F201; (* < 61953 - MG6ILAM *)
    PGN_MOTOR_GENERATOR_6_INVERTER_LIMITS_ACTIVE_DC_SIDE : UDINT := UDINT#16#F202; (* < 61954 - MG6ILADC *)
    PGN_MOTOR_GENERATOR_6_INVERTER_LOW_VOLTAGE : UDINT := UDINT#16#F203; (* < 61955 - MG6ILV *)
    PGN_MOTOR_GENERATOR_6_INVERTER_STATUS_2 : UDINT := UDINT#16#F204; (* < 61956 - MG6IS2 *)
    PGN_MOTOR_GENERATOR_6_INVERTER_RATE_LIMITS_ACTIVE_1 : UDINT := UDINT#16#F205; (* < 61957 - MG6IRLA1 *)
    PGN_BLIND_SPOT_DETECTION_1 : UDINT := UDINT#16#F206; (* < 61958 - BSD1 *)
    PGN_WINCH_INFORMATION_1 : UDINT := UDINT#16#F207; (* < 61959 - WINCH1 *)
    PGN_MOTOR_GENERATOR_3_INVERTER_CONTROL : UDINT := UDINT#16#F208; (* < 61960 - MG3IC *)
    PGN_MOTOR_GENERATOR_3_INVERTER_RATE_LIMITS_REQUEST_1 : UDINT := UDINT#16#F209; (* < 61961 - MG3IRLR1 *)
    PGN_MOTOR_GENERATOR_4_INVERTER_CONTROL : UDINT := UDINT#16#F20A; (* < 61962 - MG4IC *)
    PGN_MOTOR_GENERATOR_4_INVERTER_RATE_LIMITS_REQUEST_1 : UDINT := UDINT#16#F20B; (* < 61963 - MG4IRLR1 *)
    PGN_MOTOR_GENERATOR_5_INVERTER_CONTROL : UDINT := UDINT#16#F20C; (* < 61964 - MG5IC *)
    PGN_MOTOR_GENERATOR_5_INVERTER_RATE_LIMITS_REQUEST_1 : UDINT := UDINT#16#F20D; (* < 61965 - MG5IRLR1 *)
    PGN_MOTOR_GENERATOR_6_INVERTER_CONTROL : UDINT := UDINT#16#F20E; (* < 61966 - MG6IC *)
    PGN_MOTOR_GENERATOR_6_INVERTER_RATE_LIMITS_REQUEST_1 : UDINT := UDINT#16#F20F; (* < 61967 - MG6IRLR1 *)
    PGN_COLLISION_AVOIDANCE_SYSTEM_1 : UDINT := UDINT#16#F210; (* < 61968 - CXD1 *)
    PGN_COLLISION_AVOIDANCE_SYSTEM_2 : UDINT := UDINT#16#F211; (* < 61969 - CXD2 *)
    PGN_HIGH_VOLTAGE_ENERGY_STORAGE_PACK_7_STATUS_2 : UDINT := UDINT#16#F214; (* < 61972 - HVESP7S2 *)
    PGN_HIGH_VOLTAGE_ENERGY_STORAGE_PACK_7_DATA_1 : UDINT := UDINT#16#F215; (* < 61973 - HVESP7D1 *)
    PGN_HIGH_VOLTAGE_ENERGY_STORAGE_PACK_7_DATA_2 : UDINT := UDINT#16#F216; (* < 61974 - HVESP7D2 *)
    PGN_HIGH_VOLTAGE_ENERGY_STORAGE_PACK_7_DATA_3 : UDINT := UDINT#16#F217; (* < 61975 - HVESP7D3 *)
    PGN_HIGH_VOLTAGE_ENERGY_STORAGE_PACK_7_DATA_4 : UDINT := UDINT#16#F218; (* < 61976 - HVESP7D4 *)
    PGN_HIGH_VOLTAGE_ENERGY_STORAGE_PACK_7_DATA_5 : UDINT := UDINT#16#F219; (* < 61977 - HVESP7D5 *)
    PGN_HIGH_VOLTAGE_ENERGY_STORAGE_PACK_7_DATA_6 : UDINT := UDINT#16#F21A; (* < 61978 - HVESP7D6 *)
    PGN_HIGH_VOLTAGE_ENERGY_STORAGE_PACK_7_STATUS_1 : UDINT := UDINT#16#F21B; (* < 61979 - HVESP7S1 *)
    PGN_HIGH_VOLTAGE_ENERGY_STORAGE_PACK_7_DATA_7 : UDINT := UDINT#16#F21C; (* < 61980 - HVESP7D7 *)
    PGN_HIGH_VOLTAGE_ENERGY_STORAGE_PACK_7_MODULE_STATUS_1 : UDINT := UDINT#16#F21D; (* < 61981 - HVESP7MS1 *)
    PGN_HIGH_VOLTAGE_ENERGY_STORAGE_PACK_7_THERMAL_MANAGEMENT_SYSTEM_STATUS_1 : UDINT := UDINT#16#F21E; (* < 61982 - HVESP7TS1 *)
    PGN_HIGH_VOLTAGE_ENERGY_STORAGE_PACK_7_DATA_8 : UDINT := UDINT#16#F21F; (* < 61983 - HVESP7D8 *)
    PGN_HIGH_VOLTAGE_ENERGY_STORAGE_PACK_7_DATA_9 : UDINT := UDINT#16#F220; (* < 61984 - HVESP7D9 *)
    PGN_HIGH_VOLTAGE_ENERGY_STORAGE_PACK_7_DATA_10 : UDINT := UDINT#16#F221; (* < 61985 - HVESP7D10 *)
    PGN_HIGH_VOLTAGE_ENERGY_STORAGE_PACK_7_DATA_11 : UDINT := UDINT#16#F222; (* < 61986 - HVESP7D11 *)
    PGN_HIGH_VOLTAGE_ENERGY_STORAGE_PACK_8_STATUS_2 : UDINT := UDINT#16#F223; (* < 61987 - HVESP8S2 *)
    PGN_HIGH_VOLTAGE_ENERGY_STORAGE_PACK_8_DATA_1 : UDINT := UDINT#16#F224; (* < 61988 - HVESP8D1 *)
    PGN_HIGH_VOLTAGE_ENERGY_STORAGE_PACK_8_DATA_2 : UDINT := UDINT#16#F225; (* < 61989 - HVESP8D2 *)
    PGN_HIGH_VOLTAGE_ENERGY_STORAGE_PACK_8_DATA_3 : UDINT := UDINT#16#F226; (* < 61990 - HVESP8D3 *)
    PGN_HIGH_VOLTAGE_ENERGY_STORAGE_PACK_8_DATA_4 : UDINT := UDINT#16#F227; (* < 61991 - HVESP8D4 *)
    PGN_HIGH_VOLTAGE_ENERGY_STORAGE_PACK_8_DATA_5 : UDINT := UDINT#16#F228; (* < 61992 - HVESP8D5 *)
    PGN_HIGH_VOLTAGE_ENERGY_STORAGE_PACK_8_DATA_6 : UDINT := UDINT#16#F229; (* < 61993 - HVESP8D6 *)
    PGN_HIGH_VOLTAGE_ENERGY_STORAGE_PACK_8_STATUS_1 : UDINT := UDINT#16#F22A; (* < 61994 - HVESP8S1 *)
    PGN_HIGH_VOLTAGE_ENERGY_STORAGE_PACK_8_DATA_7 : UDINT := UDINT#16#F22B; (* < 61995 - HVESP8D7 *)
    PGN_HIGH_VOLTAGE_ENERGY_STORAGE_PACK_8_MODULE_STATUS_1 : UDINT := UDINT#16#F22C; (* < 61996 - HVESP8MS1 *)
    PGN_HIGH_VOLTAGE_ENERGY_STORAGE_PACK_8_THERMAL_MANAGEMENT_SYSTEM_STATUS_1 : UDINT := UDINT#16#F22D; (* < 61997 - HVESP8TS1 *)
    PGN_HIGH_VOLTAGE_ENERGY_STORAGE_PACK_8_DATA_8 : UDINT := UDINT#16#F22E; (* < 61998 - HVESP8D8 *)
    PGN_HIGH_VOLTAGE_ENERGY_STORAGE_PACK_8_DATA_9 : UDINT := UDINT#16#F22F; (* < 61999 - HVESP8D9 *)
    PGN_HIGH_VOLTAGE_ENERGY_STORAGE_PACK_8_DATA_10 : UDINT := UDINT#16#F230; (* < 62000 - HVESP8D10 *)
    PGN_HIGH_VOLTAGE_ENERGY_STORAGE_PACK_8_DATA_11 : UDINT := UDINT#16#F231; (* < 62001 - HVESP8D11 *)
    PGN_HIGH_VOLTAGE_ENERGY_STORAGE_PACK_9_STATUS_2 : UDINT := UDINT#16#F232; (* < 62002 - HVESP9S2 *)
    PGN_HIGH_VOLTAGE_ENERGY_STORAGE_PACK_9_DATA_1 : UDINT := UDINT#16#F233; (* < 62003 - HVESP9D1 *)
    PGN_HIGH_VOLTAGE_ENERGY_STORAGE_PACK_9_DATA_2 : UDINT := UDINT#16#F234; (* < 62004 - HVESP9D2 *)
    PGN_HIGH_VOLTAGE_ENERGY_STORAGE_PACK_9_DATA_3 : UDINT := UDINT#16#F235; (* < 62005 - HVESP9D3 *)
    PGN_HIGH_VOLTAGE_ENERGY_STORAGE_PACK_9_DATA_4 : UDINT := UDINT#16#F236; (* < 62006 - HVESP9D4 *)
    PGN_HIGH_VOLTAGE_ENERGY_STORAGE_PACK_9_DATA_5 : UDINT := UDINT#16#F237; (* < 62007 - HVESP9D5 *)
    PGN_HIGH_VOLTAGE_ENERGY_STORAGE_PACK_9_DATA_6 : UDINT := UDINT#16#F238; (* < 62008 - HVESP9D6 *)
    PGN_HIGH_VOLTAGE_ENERGY_STORAGE_PACK_9_STATUS_1 : UDINT := UDINT#16#F239; (* < 62009 - HVESP9S1 *)
    PGN_HIGH_VOLTAGE_ENERGY_STORAGE_PACK_9_DATA_7 : UDINT := UDINT#16#F23A; (* < 62010 - HVESP9D7 *)
    PGN_HIGH_VOLTAGE_ENERGY_STORAGE_PACK_9_MODULE_STATUS_1 : UDINT := UDINT#16#F23B; (* < 62011 - HVESP9MS1 *)
    PGN_HIGH_VOLTAGE_ENERGY_STORAGE_PACK_9_THERMAL_MANAGEMENT_SYSTEM_STATUS_1 : UDINT := UDINT#16#F23C; (* < 62012 - HVESP9TS1 *)
    PGN_HIGH_VOLTAGE_ENERGY_STORAGE_PACK_9_DATA_8 : UDINT := UDINT#16#F23D; (* < 62013 - HVESP9D8 *)
    PGN_HIGH_VOLTAGE_ENERGY_STORAGE_PACK_9_DATA_9 : UDINT := UDINT#16#F23E; (* < 62014 - HVESP9D9 *)
    PGN_HIGH_VOLTAGE_ENERGY_STORAGE_PACK_9_DATA_10 : UDINT := UDINT#16#F23F; (* < 62015 - HVESP9D10 *)
    PGN_HIGH_VOLTAGE_ENERGY_STORAGE_PACK_9_DATA_11 : UDINT := UDINT#16#F240; (* < 62016 - HVESP9D11 *)
    PGN_HIGH_VOLTAGE_ENERGY_STORAGE_PACK_10_STATUS_2 : UDINT := UDINT#16#F241; (* < 62017 - HVESP10S2 *)
    PGN_HIGH_VOLTAGE_ENERGY_STORAGE_PACK_10_DATA_1 : UDINT := UDINT#16#F242; (* < 62018 - HVESP10D1 *)
    PGN_HIGH_VOLTAGE_ENERGY_STORAGE_PACK_10_DATA_2 : UDINT := UDINT#16#F243; (* < 62019 - HVESP10D2 *)
    PGN_HIGH_VOLTAGE_ENERGY_STORAGE_PACK_10_DATA_3 : UDINT := UDINT#16#F244; (* < 62020 - HVESP10D3 *)
    PGN_HIGH_VOLTAGE_ENERGY_STORAGE_PACK_10_DATA_4 : UDINT := UDINT#16#F245; (* < 62021 - HVESP10D4 *)
    PGN_HIGH_VOLTAGE_ENERGY_STORAGE_PACK_10_DATA_5 : UDINT := UDINT#16#F246; (* < 62022 - HVESP10D5 *)
    PGN_HIGH_VOLTAGE_ENERGY_STORAGE_PACK_10_DATA_6 : UDINT := UDINT#16#F247; (* < 62023 - HVESP10D6 *)
    PGN_HIGH_VOLTAGE_ENERGY_STORAGE_PACK_10_STATUS_1 : UDINT := UDINT#16#F248; (* < 62024 - HVESP10S1 *)
    PGN_HIGH_VOLTAGE_ENERGY_STORAGE_PACK_10_DATA_7 : UDINT := UDINT#16#F249; (* < 62025 - HVESP10D7 *)
    PGN_HIGH_VOLTAGE_ENERGY_STORAGE_PACK_10_MODULE_STATUS_1 : UDINT := UDINT#16#F24A; (* < 62026 - HVESP10MS1 *)
    PGN_HIGH_VOLTAGE_ENERGY_STORAGE_PACK_10_THERMAL_MANAGEMENT_SYSTEM_STATUS_1 : UDINT := UDINT#16#F24B; (* < 62027 - HVESP10TS1 *)
    PGN_HIGH_VOLTAGE_ENERGY_STORAGE_PACK_10_DATA_8 : UDINT := UDINT#16#F24C; (* < 62028 - HVESP10D8 *)
    PGN_HIGH_VOLTAGE_ENERGY_STORAGE_PACK_10_DATA_9 : UDINT := UDINT#16#F24D; (* < 62029 - HVESP10D9 *)
    PGN_HIGH_VOLTAGE_ENERGY_STORAGE_PACK_10_DATA_10 : UDINT := UDINT#16#F24E; (* < 62030 - HVESP10D10 *)
    PGN_HIGH_VOLTAGE_ENERGY_STORAGE_PACK_10_DATA_11 : UDINT := UDINT#16#F24F; (* < 62031 - HVESP10D11 *)
    PGN_ELECTRONIC_AUXILIARY_TRANSMISSION_CONTROLLER_1 : UDINT := UDINT#16#F250; (* < 62032 - EATC1 *)
    PGN_HIGH_VOLTAGE_ENERGY_STORAGE_PACK_11_STATUS_2 : UDINT := UDINT#16#F251; (* < 62033 - HVESP11S2 *)
    PGN_HIGH_VOLTAGE_ENERGY_STORAGE_PACK_11_DATA_1 : UDINT := UDINT#16#F252; (* < 62034 - HVESP11D1 *)
    PGN_HIGH_VOLTAGE_ENERGY_STORAGE_PACK_11_DATA_2 : UDINT := UDINT#16#F253; (* < 62035 - HVESP11D2 *)
    PGN_HIGH_VOLTAGE_ENERGY_STORAGE_PACK_11_DATA_3 : UDINT := UDINT#16#F254; (* < 62036 - HVESP11D3 *)
    PGN_HIGH_VOLTAGE_ENERGY_STORAGE_PACK_11_DATA_4 : UDINT := UDINT#16#F255; (* < 62037 - HVESP11D4 *)
    PGN_HIGH_VOLTAGE_ENERGY_STORAGE_PACK_11_DATA_5 : UDINT := UDINT#16#F256; (* < 62038 - HVESP11D5 *)
    PGN_HIGH_VOLTAGE_ENERGY_STORAGE_PACK_11_DATA_6 : UDINT := UDINT#16#F257; (* < 62039 - HVESP11D6 *)
    PGN_HIGH_VOLTAGE_ENERGY_STORAGE_PACK_11_STATUS_1 : UDINT := UDINT#16#F258; (* < 62040 - HVESP11S1 *)
    PGN_HIGH_VOLTAGE_ENERGY_STORAGE_PACK_11_DATA_7 : UDINT := UDINT#16#F259; (* < 62041 - HVESP11D7 *)
    PGN_HIGH_VOLTAGE_ENERGY_STORAGE_PACK_11_MODULE_STATUS_1 : UDINT := UDINT#16#F25A; (* < 62042 - HVESP11MS1 *)
    PGN_HIGH_VOLTAGE_ENERGY_STORAGE_PACK_11_THERMAL_MANAGEMENT_SYSTEM_STATUS_1 : UDINT := UDINT#16#F25B; (* < 62043 - HVESP11TS1 *)
    PGN_HIGH_VOLTAGE_ENERGY_STORAGE_PACK_11_DATA_8 : UDINT := UDINT#16#F25C; (* < 62044 - HVESP11D8 *)
    PGN_HIGH_VOLTAGE_ENERGY_STORAGE_PACK_11_DATA_9 : UDINT := UDINT#16#F25D; (* < 62045 - HVESP11D9 *)
    PGN_HIGH_VOLTAGE_ENERGY_STORAGE_PACK_11_DATA_10 : UDINT := UDINT#16#F25E; (* < 62046 - HVESP11D10 *)
    PGN_HIGH_VOLTAGE_ENERGY_STORAGE_PACK_11_DATA_11 : UDINT := UDINT#16#F25F; (* < 62047 - HVESP11D11 *)
    PGN_HIGH_VOLTAGE_ENERGY_STORAGE_PACK_12_STATUS_2 : UDINT := UDINT#16#F260; (* < 62048 - HVESP12S2 *)
    PGN_HIGH_VOLTAGE_ENERGY_STORAGE_PACK_12_DATA_1 : UDINT := UDINT#16#F261; (* < 62049 - HVESP12D1 *)
    PGN_HIGH_VOLTAGE_ENERGY_STORAGE_PACK_12_DATA_2 : UDINT := UDINT#16#F262; (* < 62050 - HVESP12D2 *)
    PGN_HIGH_VOLTAGE_ENERGY_STORAGE_PACK_12_DATA_3 : UDINT := UDINT#16#F263; (* < 62051 - HVESP12D3 *)
    PGN_HIGH_VOLTAGE_ENERGY_STORAGE_PACK_12_DATA_4 : UDINT := UDINT#16#F264; (* < 62052 - HVESP12D4 *)
    PGN_HIGH_VOLTAGE_ENERGY_STORAGE_PACK_12_DATA_5 : UDINT := UDINT#16#F265; (* < 62053 - HVESP12D5 *)
    PGN_HIGH_VOLTAGE_ENERGY_STORAGE_PACK_12_DATA_6 : UDINT := UDINT#16#F266; (* < 62054 - HVESP12D6 *)
    PGN_HIGH_VOLTAGE_ENERGY_STORAGE_PACK_12_STATUS_1 : UDINT := UDINT#16#F267; (* < 62055 - HVESP12S1 *)
    PGN_HIGH_VOLTAGE_ENERGY_STORAGE_PACK_12_DATA_7 : UDINT := UDINT#16#F268; (* < 62056 - HVESP12D7 *)
    PGN_HIGH_VOLTAGE_ENERGY_STORAGE_PACK_12_MODULE_STATUS_1 : UDINT := UDINT#16#F269; (* < 62057 - HVESP12MS1 *)
    PGN_HIGH_VOLTAGE_ENERGY_STORAGE_PACK_12_THERMAL_MANAGEMENT_SYSTEM_STATUS_1 : UDINT := UDINT#16#F26A; (* < 62058 - HVESP12TS1 *)
    PGN_HIGH_VOLTAGE_ENERGY_STORAGE_PACK_12_DATA_8 : UDINT := UDINT#16#F26B; (* < 62059 - HVESP12D8 *)
    PGN_HIGH_VOLTAGE_ENERGY_STORAGE_PACK_12_DATA_9 : UDINT := UDINT#16#F26C; (* < 62060 - HVESP12D9 *)
    PGN_HIGH_VOLTAGE_ENERGY_STORAGE_PACK_12_DATA_10 : UDINT := UDINT#16#F26D; (* < 62061 - HVESP12D10 *)
    PGN_HIGH_VOLTAGE_ENERGY_STORAGE_PACK_12_DATA_11 : UDINT := UDINT#16#F26E; (* < 62062 - HVESP12D11 *)
    PGN_HIGH_VOLTAGE_ENERGY_STORAGE_PACK_13_STATUS_2 : UDINT := UDINT#16#F26F; (* < 62063 - HVESP13S2 *)
    PGN_HIGH_VOLTAGE_ENERGY_STORAGE_PACK_13_DATA_1 : UDINT := UDINT#16#F270; (* < 62064 - HVESP13D1 *)
    PGN_HIGH_VOLTAGE_ENERGY_STORAGE_PACK_13_DATA_2 : UDINT := UDINT#16#F271; (* < 62065 - HVESP13D2 *)
    PGN_HIGH_VOLTAGE_ENERGY_STORAGE_PACK_13_DATA_3 : UDINT := UDINT#16#F272; (* < 62066 - HVESP13D3 *)
    PGN_HIGH_VOLTAGE_ENERGY_STORAGE_PACK_13_DATA_4 : UDINT := UDINT#16#F273; (* < 62067 - HVESP13D4 *)
    PGN_HIGH_VOLTAGE_ENERGY_STORAGE_PACK_13_DATA_5 : UDINT := UDINT#16#F274; (* < 62068 - HVESP13D5 *)
    PGN_HIGH_VOLTAGE_ENERGY_STORAGE_PACK_13_DATA_6 : UDINT := UDINT#16#F275; (* < 62069 - HVESP13D6 *)
    PGN_HIGH_VOLTAGE_ENERGY_STORAGE_PACK_13_STATUS_1 : UDINT := UDINT#16#F276; (* < 62070 - HVESP13S1 *)
    PGN_HIGH_VOLTAGE_ENERGY_STORAGE_PACK_13_DATA_7 : UDINT := UDINT#16#F277; (* < 62071 - HVESP13D7 *)
    PGN_HIGH_VOLTAGE_ENERGY_STORAGE_PACK_13_MODULE_STATUS_1 : UDINT := UDINT#16#F278; (* < 62072 - HVESP13MS1 *)
    PGN_HIGH_VOLTAGE_ENERGY_STORAGE_PACK_13_THERMAL_MANAGEMENT_SYSTEM_STATUS_1 : UDINT := UDINT#16#F279; (* < 62073 - HVESP13TS1 *)
    PGN_HIGH_VOLTAGE_ENERGY_STORAGE_PACK_13_DATA_8 : UDINT := UDINT#16#F27A; (* < 62074 - HVESP13D8 *)
    PGN_HIGH_VOLTAGE_ENERGY_STORAGE_PACK_13_DATA_9 : UDINT := UDINT#16#F27B; (* < 62075 - HVESP13D9 *)
    PGN_HIGH_VOLTAGE_ENERGY_STORAGE_PACK_13_DATA_10 : UDINT := UDINT#16#F27C; (* < 62076 - HVESP13D10 *)
    PGN_HIGH_VOLTAGE_ENERGY_STORAGE_PACK_13_DATA_11 : UDINT := UDINT#16#F27D; (* < 62077 - HVESP13D11 *)
    PGN_HIGH_VOLTAGE_ENERGY_STORAGE_PACK_14_STATUS_2 : UDINT := UDINT#16#F27E; (* < 62078 - HVESP14S2 *)
    PGN_HIGH_VOLTAGE_ENERGY_STORAGE_PACK_14_DATA_1 : UDINT := UDINT#16#F27F; (* < 62079 - HVESP14D1 *)
    PGN_HIGH_VOLTAGE_ENERGY_STORAGE_PACK_14_DATA_2 : UDINT := UDINT#16#F280; (* < 62080 - HVESP14D2 *)
    PGN_HIGH_VOLTAGE_ENERGY_STORAGE_PACK_14_DATA_3 : UDINT := UDINT#16#F281; (* < 62081 - HVESP14D3 *)
    PGN_HIGH_VOLTAGE_ENERGY_STORAGE_PACK_14_DATA_4 : UDINT := UDINT#16#F282; (* < 62082 - HVESP14D4 *)
    PGN_HIGH_VOLTAGE_ENERGY_STORAGE_PACK_14_DATA_5 : UDINT := UDINT#16#F283; (* < 62083 - HVESP14D5 *)
    PGN_HIGH_VOLTAGE_ENERGY_STORAGE_PACK_14_DATA_6 : UDINT := UDINT#16#F284; (* < 62084 - HVESP14D6 *)
    PGN_HIGH_VOLTAGE_ENERGY_STORAGE_PACK_14_STATUS_1 : UDINT := UDINT#16#F285; (* < 62085 - HVESP14S1 *)
    PGN_HIGH_VOLTAGE_ENERGY_STORAGE_PACK_14_DATA_7 : UDINT := UDINT#16#F286; (* < 62086 - HVESP14D7 *)
    PGN_HIGH_VOLTAGE_ENERGY_STORAGE_PACK_14_MODULE_STATUS_1 : UDINT := UDINT#16#F287; (* < 62087 - HVESP14MS1 *)
    PGN_HIGH_VOLTAGE_ENERGY_STORAGE_PACK_14_THERMAL_MANAGEMENT_SYSTEM_STATUS_1 : UDINT := UDINT#16#F288; (* < 62088 - HVESP14TS1 *)
    PGN_HIGH_VOLTAGE_ENERGY_STORAGE_PACK_14_DATA_8 : UDINT := UDINT#16#F289; (* < 62089 - HVESP14D8 *)
    PGN_HIGH_VOLTAGE_ENERGY_STORAGE_PACK_14_DATA_9 : UDINT := UDINT#16#F28A; (* < 62090 - HVESP14D9 *)
    PGN_HIGH_VOLTAGE_ENERGY_STORAGE_PACK_14_DATA_10 : UDINT := UDINT#16#F28B; (* < 62091 - HVESP14D10 *)
    PGN_HIGH_VOLTAGE_ENERGY_STORAGE_PACK_14_DATA_11 : UDINT := UDINT#16#F28C; (* < 62092 - HVESP14D11 *)
    PGN_HIGH_VOLTAGE_ENERGY_STORAGE_PACK_15_STATUS_2 : UDINT := UDINT#16#F28D; (* < 62093 - HVESP15S2 *)
    PGN_HIGH_VOLTAGE_ENERGY_STORAGE_PACK_15_DATA_1 : UDINT := UDINT#16#F28E; (* < 62094 - HVESP15D1 *)
    PGN_HIGH_VOLTAGE_ENERGY_STORAGE_PACK_15_DATA_2 : UDINT := UDINT#16#F28F; (* < 62095 - HVESP15D2 *)
    PGN_HIGH_VOLTAGE_ENERGY_STORAGE_PACK_15_DATA_3 : UDINT := UDINT#16#F290; (* < 62096 - HVESP15D3 *)
    PGN_HIGH_VOLTAGE_ENERGY_STORAGE_PACK_15_DATA_4 : UDINT := UDINT#16#F291; (* < 62097 - HVESP15D4 *)
    PGN_HIGH_VOLTAGE_ENERGY_STORAGE_PACK_15_DATA_5 : UDINT := UDINT#16#F292; (* < 62098 - HVESP15D5 *)
    PGN_HIGH_VOLTAGE_ENERGY_STORAGE_PACK_15_DATA_6 : UDINT := UDINT#16#F293; (* < 62099 - HVESP15D6 *)
    PGN_HIGH_VOLTAGE_ENERGY_STORAGE_PACK_15_STATUS_1 : UDINT := UDINT#16#F294; (* < 62100 - HVESP15S1 *)
    PGN_HIGH_VOLTAGE_ENERGY_STORAGE_PACK_15_DATA_7 : UDINT := UDINT#16#F295; (* < 62101 - HVESP15D7 *)
    PGN_HIGH_VOLTAGE_ENERGY_STORAGE_PACK_15_MODULE_STATUS_1 : UDINT := UDINT#16#F296; (* < 62102 - HVESP15MS1 *)
    PGN_HIGH_VOLTAGE_ENERGY_STORAGE_PACK_15_THERMAL_MANAGEMENT_SYSTEM_STATUS_1 : UDINT := UDINT#16#F297; (* < 62103 - HVESP15TS1 *)
    PGN_HIGH_VOLTAGE_ENERGY_STORAGE_PACK_15_DATA_8 : UDINT := UDINT#16#F298; (* < 62104 - HVESP15D8 *)
    PGN_HIGH_VOLTAGE_ENERGY_STORAGE_PACK_15_DATA_9 : UDINT := UDINT#16#F299; (* < 62105 - HVESP15D9 *)
    PGN_HIGH_VOLTAGE_ENERGY_STORAGE_PACK_15_DATA_10 : UDINT := UDINT#16#F29A; (* < 62106 - HVESP15D10 *)
    PGN_HIGH_VOLTAGE_ENERGY_STORAGE_PACK_15_DATA_11 : UDINT := UDINT#16#F29B; (* < 62107 - HVESP15D11 *)
    PGN_HIGH_VOLTAGE_ENERGY_STORAGE_PACK_16_STATUS_2 : UDINT := UDINT#16#F29C; (* < 62108 - HVESP16S2 *)
    PGN_HIGH_VOLTAGE_ENERGY_STORAGE_PACK_16_DATA_1 : UDINT := UDINT#16#F29D; (* < 62109 - HVESP16D1 *)
    PGN_HIGH_VOLTAGE_ENERGY_STORAGE_PACK_16_DATA_2 : UDINT := UDINT#16#F29E; (* < 62110 - HVESP16D2 *)
    PGN_HIGH_VOLTAGE_ENERGY_STORAGE_PACK_16_DATA_3 : UDINT := UDINT#16#F29F; (* < 62111 - HVESP16D3 *)
    PGN_HIGH_VOLTAGE_ENERGY_STORAGE_PACK_16_DATA_4 : UDINT := UDINT#16#F2A0; (* < 62112 - HVESP16D4 *)
    PGN_HIGH_VOLTAGE_ENERGY_STORAGE_PACK_16_DATA_5 : UDINT := UDINT#16#F2A1; (* < 62113 - HVESP16D5 *)
    PGN_HIGH_VOLTAGE_ENERGY_STORAGE_PACK_16_DATA_6 : UDINT := UDINT#16#F2A2; (* < 62114 - HVESP16D6 *)
    PGN_HIGH_VOLTAGE_ENERGY_STORAGE_PACK_16_STATUS_1 : UDINT := UDINT#16#F2A3; (* < 62115 - HVESP16S1 *)
    PGN_HIGH_VOLTAGE_ENERGY_STORAGE_PACK_16_DATA_7 : UDINT := UDINT#16#F2A4; (* < 62116 - HVESP16D7 *)
    PGN_HIGH_VOLTAGE_ENERGY_STORAGE_PACK_16_MODULE_STATUS_1 : UDINT := UDINT#16#F2A5; (* < 62117 - HVESP16MS1 *)
    PGN_HIGH_VOLTAGE_ENERGY_STORAGE_PACK_16_THERMAL_MANAGEMENT_SYSTEM_STATUS_1 : UDINT := UDINT#16#F2A6; (* < 62118 - HVESP16TS1 *)
    PGN_HIGH_VOLTAGE_ENERGY_STORAGE_PACK_16_DATA_8 : UDINT := UDINT#16#F2A7; (* < 62119 - HVESP16D8 *)
    PGN_HIGH_VOLTAGE_ENERGY_STORAGE_PACK_16_DATA_9 : UDINT := UDINT#16#F2A8; (* < 62120 - HVESP16D9 *)
    PGN_HIGH_VOLTAGE_ENERGY_STORAGE_PACK_16_DATA_10 : UDINT := UDINT#16#F2A9; (* < 62121 - HVESP16D10 *)
    PGN_HIGH_VOLTAGE_ENERGY_STORAGE_PACK_16_DATA_11 : UDINT := UDINT#16#F2AA; (* < 62122 - HVESP16D11 *)
    PGN_HIGH_VOLTAGE_ENERGY_STORAGE_PACK_17_STATUS_2 : UDINT := UDINT#16#F2AB; (* < 62123 - HVESP17S2 *)
    PGN_HIGH_VOLTAGE_ENERGY_STORAGE_PACK_17_DATA_1 : UDINT := UDINT#16#F2AC; (* < 62124 - HVESP17D1 *)
    PGN_HIGH_VOLTAGE_ENERGY_STORAGE_PACK_17_DATA_2 : UDINT := UDINT#16#F2AD; (* < 62125 - HVESP17D2 *)
    PGN_HIGH_VOLTAGE_ENERGY_STORAGE_PACK_17_DATA_3 : UDINT := UDINT#16#F2AE; (* < 62126 - HVESP17D3 *)
    PGN_HIGH_VOLTAGE_ENERGY_STORAGE_PACK_17_DATA_4 : UDINT := UDINT#16#F2AF; (* < 62127 - HVESP17D4 *)
    PGN_HIGH_VOLTAGE_ENERGY_STORAGE_PACK_17_DATA_5 : UDINT := UDINT#16#F2B0; (* < 62128 - HVESP17D5 *)
    PGN_HIGH_VOLTAGE_ENERGY_STORAGE_PACK_17_DATA_6 : UDINT := UDINT#16#F2B1; (* < 62129 - HVESP17D6 *)
    PGN_HIGH_VOLTAGE_ENERGY_STORAGE_PACK_17_STATUS_1 : UDINT := UDINT#16#F2B2; (* < 62130 - HVESP17S1 *)
    PGN_HIGH_VOLTAGE_ENERGY_STORAGE_PACK_17_DATA_7 : UDINT := UDINT#16#F2B3; (* < 62131 - HVESP17D7 *)
    PGN_HIGH_VOLTAGE_ENERGY_STORAGE_PACK_17_MODULE_STATUS_1 : UDINT := UDINT#16#F2B4; (* < 62132 - HVESP17MS1 *)
    PGN_HIGH_VOLTAGE_ENERGY_STORAGE_PACK_17_THERMAL_MANAGEMENT_SYSTEM_STATUS_1 : UDINT := UDINT#16#F2B5; (* < 62133 - HVESP17TS1 *)
    PGN_HIGH_VOLTAGE_ENERGY_STORAGE_PACK_17_DATA_8 : UDINT := UDINT#16#F2B6; (* < 62134 - HVESP17D8 *)
    PGN_HIGH_VOLTAGE_ENERGY_STORAGE_PACK_17_DATA_9 : UDINT := UDINT#16#F2B7; (* < 62135 - HVESP17D9 *)
    PGN_HIGH_VOLTAGE_ENERGY_STORAGE_PACK_17_DATA_10 : UDINT := UDINT#16#F2B8; (* < 62136 - HVESP17D10 *)
    PGN_HIGH_VOLTAGE_ENERGY_STORAGE_PACK_17_DATA_11 : UDINT := UDINT#16#F2B9; (* < 62137 - HVESP17D11 *)
    PGN_HIGH_VOLTAGE_ENERGY_STORAGE_PACK_18_STATUS_2 : UDINT := UDINT#16#F2BA; (* < 62138 - HVESP18S2 *)
    PGN_HIGH_VOLTAGE_ENERGY_STORAGE_PACK_18_DATA_1 : UDINT := UDINT#16#F2BB; (* < 62139 - HVESP18D1 *)
    PGN_HIGH_VOLTAGE_ENERGY_STORAGE_PACK_18_DATA_2 : UDINT := UDINT#16#F2BC; (* < 62140 - HVESP18D2 *)
    PGN_HIGH_VOLTAGE_ENERGY_STORAGE_PACK_18_DATA_3 : UDINT := UDINT#16#F2BD; (* < 62141 - HVESP18D3 *)
    PGN_HIGH_VOLTAGE_ENERGY_STORAGE_PACK_18_DATA_4 : UDINT := UDINT#16#F2BE; (* < 62142 - HVESP18D4 *)
    PGN_HIGH_VOLTAGE_ENERGY_STORAGE_PACK_18_DATA_5 : UDINT := UDINT#16#F2BF; (* < 62143 - HVESP18D5 *)
    PGN_HIGH_VOLTAGE_ENERGY_STORAGE_PACK_18_DATA_6 : UDINT := UDINT#16#F2C0; (* < 62144 - HVESP18D6 *)
    PGN_HIGH_VOLTAGE_ENERGY_STORAGE_PACK_18_STATUS_1 : UDINT := UDINT#16#F2C1; (* < 62145 - HVESP18S1 *)
    PGN_HIGH_VOLTAGE_ENERGY_STORAGE_PACK_18_DATA_7 : UDINT := UDINT#16#F2C2; (* < 62146 - HVESP18D7 *)
    PGN_HIGH_VOLTAGE_ENERGY_STORAGE_PACK_18_MODULE_STATUS_1 : UDINT := UDINT#16#F2C3; (* < 62147 - HVESP18MS1 *)
    PGN_HIGH_VOLTAGE_ENERGY_STORAGE_PACK_18_THERMAL_MANAGEMENT_SYSTEM_STATUS_1 : UDINT := UDINT#16#F2C4; (* < 62148 - HVESP18TS1 *)
    PGN_HIGH_VOLTAGE_ENERGY_STORAGE_PACK_18_DATA_8 : UDINT := UDINT#16#F2C5; (* < 62149 - HVESP18D8 *)
    PGN_HIGH_VOLTAGE_ENERGY_STORAGE_PACK_18_DATA_9 : UDINT := UDINT#16#F2C6; (* < 62150 - HVESP18D9 *)
    PGN_HIGH_VOLTAGE_ENERGY_STORAGE_PACK_18_DATA_10 : UDINT := UDINT#16#F2C7; (* < 62151 - HVESP18D10 *)
    PGN_HIGH_VOLTAGE_ENERGY_STORAGE_PACK_18_DATA_11 : UDINT := UDINT#16#F2C8; (* < 62152 - HVESP18D11 *)
    PGN_HIGH_VOLTAGE_ENERGY_STORAGE_PACK_19_STATUS_2 : UDINT := UDINT#16#F2C9; (* < 62153 - HVESP19S2 *)
    PGN_HIGH_VOLTAGE_ENERGY_STORAGE_PACK_19_DATA_1 : UDINT := UDINT#16#F2CA; (* < 62154 - HVESP19D1 *)
    PGN_HIGH_VOLTAGE_ENERGY_STORAGE_PACK_19_DATA_2 : UDINT := UDINT#16#F2CB; (* < 62155 - HVESP19D2 *)
    PGN_HIGH_VOLTAGE_ENERGY_STORAGE_PACK_19_DATA_3 : UDINT := UDINT#16#F2CC; (* < 62156 - HVESP19D3 *)
    PGN_HIGH_VOLTAGE_ENERGY_STORAGE_PACK_19_DATA_4 : UDINT := UDINT#16#F2CD; (* < 62157 - HVESP19D4 *)
    PGN_HIGH_VOLTAGE_ENERGY_STORAGE_PACK_19_DATA_5 : UDINT := UDINT#16#F2CE; (* < 62158 - HVESP19D5 *)
    PGN_HIGH_VOLTAGE_ENERGY_STORAGE_PACK_19_DATA_6 : UDINT := UDINT#16#F2CF; (* < 62159 - HVESP19D6 *)
    PGN_HIGH_VOLTAGE_ENERGY_STORAGE_PACK_19_STATUS_1 : UDINT := UDINT#16#F2D0; (* < 62160 - HVESP19S1 *)
    PGN_HIGH_VOLTAGE_ENERGY_STORAGE_PACK_19_DATA_7 : UDINT := UDINT#16#F2D1; (* < 62161 - HVESP19D7 *)
    PGN_HIGH_VOLTAGE_ENERGY_STORAGE_PACK_19_MODULE_STATUS_1 : UDINT := UDINT#16#F2D2; (* < 62162 - HVESP19MS1 *)
    PGN_HIGH_VOLTAGE_ENERGY_STORAGE_PACK_19_THERMAL_MANAGEMENT_SYSTEM_STATUS_1 : UDINT := UDINT#16#F2D3; (* < 62163 - HVESP19TS1 *)
    PGN_HIGH_VOLTAGE_ENERGY_STORAGE_PACK_19_DATA_8 : UDINT := UDINT#16#F2D4; (* < 62164 - HVESP19D8 *)
    PGN_HIGH_VOLTAGE_ENERGY_STORAGE_PACK_19_DATA_9 : UDINT := UDINT#16#F2D5; (* < 62165 - HVESP19D9 *)
    PGN_HIGH_VOLTAGE_ENERGY_STORAGE_PACK_19_DATA_10 : UDINT := UDINT#16#F2D6; (* < 62166 - HVESP19D10 *)
    PGN_HIGH_VOLTAGE_ENERGY_STORAGE_PACK_19_DATA_11 : UDINT := UDINT#16#F2D7; (* < 62167 - HVESP19D11 *)
    PGN_HIGH_VOLTAGE_ENERGY_STORAGE_PACK_20_STATUS_2 : UDINT := UDINT#16#F2D8; (* < 62168 - HVESP20S2 *)
    PGN_HIGH_VOLTAGE_ENERGY_STORAGE_PACK_20_DATA_1 : UDINT := UDINT#16#F2D9; (* < 62169 - HVESP20D1 *)
    PGN_HIGH_VOLTAGE_ENERGY_STORAGE_PACK_20_DATA_2 : UDINT := UDINT#16#F2DA; (* < 62170 - HVESP20D2 *)
    PGN_HIGH_VOLTAGE_ENERGY_STORAGE_PACK_20_DATA_3 : UDINT := UDINT#16#F2DB; (* < 62171 - HVESP20D3 *)
    PGN_HIGH_VOLTAGE_ENERGY_STORAGE_PACK_20_DATA_4 : UDINT := UDINT#16#F2DC; (* < 62172 - HVESP20D4 *)
    PGN_HIGH_VOLTAGE_ENERGY_STORAGE_PACK_20_DATA_5 : UDINT := UDINT#16#F2DD; (* < 62173 - HVESP20D5 *)
    PGN_HIGH_VOLTAGE_ENERGY_STORAGE_PACK_20_DATA_6 : UDINT := UDINT#16#F2DE; (* < 62174 - HVESP20D6 *)
    PGN_HIGH_VOLTAGE_ENERGY_STORAGE_PACK_20_STATUS_1 : UDINT := UDINT#16#F2DF; (* < 62175 - HVESP20S1 *)
    PGN_HIGH_VOLTAGE_ENERGY_STORAGE_PACK_20_DATA_7 : UDINT := UDINT#16#F2E0; (* < 62176 - HVESP20D7 *)
    PGN_HIGH_VOLTAGE_ENERGY_STORAGE_PACK_20_MODULE_STATUS_1 : UDINT := UDINT#16#F2E1; (* < 62177 - HVESP20MS1 *)
    PGN_HIGH_VOLTAGE_ENERGY_STORAGE_PACK_20_THERMAL_MANAGEMENT_SYSTEM_STATUS_1 : UDINT := UDINT#16#F2E2; (* < 62178 - HVESP20TS1 *)
    PGN_HIGH_VOLTAGE_ENERGY_STORAGE_PACK_20_DATA_8 : UDINT := UDINT#16#F2E3; (* < 62179 - HVESP20D8 *)
    PGN_HIGH_VOLTAGE_ENERGY_STORAGE_PACK_20_DATA_9 : UDINT := UDINT#16#F2E4; (* < 62180 - HVESP20D9 *)
    PGN_HIGH_VOLTAGE_ENERGY_STORAGE_PACK_20_DATA_10 : UDINT := UDINT#16#F2E5; (* < 62181 - HVESP20D10 *)
    PGN_HIGH_VOLTAGE_ENERGY_STORAGE_PACK_20_DATA_11 : UDINT := UDINT#16#F2E6; (* < 62182 - HVESP20D11 *)
    PGN_HIGH_VOLTAGE_ENERGY_STORAGE_PACK_21_STATUS_2 : UDINT := UDINT#16#F2E7; (* < 62183 - HVESP21S2 *)
    PGN_HIGH_VOLTAGE_ENERGY_STORAGE_PACK_21_DATA_1 : UDINT := UDINT#16#F2E8; (* < 62184 - HVESP21D1 *)
    PGN_HIGH_VOLTAGE_ENERGY_STORAGE_PACK_21_DATA_2 : UDINT := UDINT#16#F2E9; (* < 62185 - HVESP21D2 *)
    PGN_HIGH_VOLTAGE_ENERGY_STORAGE_PACK_21_DATA_3 : UDINT := UDINT#16#F2EA; (* < 62186 - HVESP21D3 *)
    PGN_HIGH_VOLTAGE_ENERGY_STORAGE_PACK_21_DATA_4 : UDINT := UDINT#16#F2EB; (* < 62187 - HVESP21D4 *)
    PGN_HIGH_VOLTAGE_ENERGY_STORAGE_PACK_21_DATA_5 : UDINT := UDINT#16#F2EC; (* < 62188 - HVESP21D5 *)
    PGN_HIGH_VOLTAGE_ENERGY_STORAGE_PACK_21_DATA_6 : UDINT := UDINT#16#F2ED; (* < 62189 - HVESP21D6 *)
    PGN_HIGH_VOLTAGE_ENERGY_STORAGE_PACK_21_STATUS_1 : UDINT := UDINT#16#F2EE; (* < 62190 - HVESP21S1 *)
    PGN_HIGH_VOLTAGE_ENERGY_STORAGE_PACK_21_DATA_7 : UDINT := UDINT#16#F2EF; (* < 62191 - HVESP21D7 *)
    PGN_HIGH_VOLTAGE_ENERGY_STORAGE_PACK_21_MODULE_STATUS_1 : UDINT := UDINT#16#F2F0; (* < 62192 - HVESP21MS1 *)
    PGN_HIGH_VOLTAGE_ENERGY_STORAGE_PACK_21_THERMAL_MANAGEMENT_SYSTEM_STATUS_1 : UDINT := UDINT#16#F2F1; (* < 62193 - HVESP21TS1 *)
    PGN_HIGH_VOLTAGE_ENERGY_STORAGE_PACK_21_DATA_8 : UDINT := UDINT#16#F2F2; (* < 62194 - HVESP21D8 *)
    PGN_HIGH_VOLTAGE_ENERGY_STORAGE_PACK_21_DATA_9 : UDINT := UDINT#16#F2F3; (* < 62195 - HVESP21D9 *)
    PGN_HIGH_VOLTAGE_ENERGY_STORAGE_PACK_21_DATA_10 : UDINT := UDINT#16#F2F4; (* < 62196 - HVESP21D10 *)
    PGN_HIGH_VOLTAGE_ENERGY_STORAGE_PACK_21_DATA_11 : UDINT := UDINT#16#F2F5; (* < 62197 - HVESP21D11 *)
    PGN_HIGH_VOLTAGE_ENERGY_STORAGE_PACK_22_STATUS_2 : UDINT := UDINT#16#F2F6; (* < 62198 - HVESP22S2 *)
    PGN_HIGH_VOLTAGE_ENERGY_STORAGE_PACK_22_DATA_1 : UDINT := UDINT#16#F2F7; (* < 62199 - HVESP22D1 *)
    PGN_HIGH_VOLTAGE_ENERGY_STORAGE_PACK_22_DATA_2 : UDINT := UDINT#16#F2F8; (* < 62200 - HVESP22D2 *)
    PGN_HIGH_VOLTAGE_ENERGY_STORAGE_PACK_22_DATA_3 : UDINT := UDINT#16#F2F9; (* < 62201 - HVESP22D3 *)
    PGN_HIGH_VOLTAGE_ENERGY_STORAGE_PACK_22_DATA_4 : UDINT := UDINT#16#F2FA; (* < 62202 - HVESP22D4 *)
    PGN_HIGH_VOLTAGE_ENERGY_STORAGE_PACK_22_DATA_5 : UDINT := UDINT#16#F2FB; (* < 62203 - HVESP22D5 *)
    PGN_HIGH_VOLTAGE_ENERGY_STORAGE_PACK_22_DATA_6 : UDINT := UDINT#16#F2FC; (* < 62204 - HVESP22D6 *)
    PGN_HIGH_VOLTAGE_ENERGY_STORAGE_PACK_22_STATUS_1 : UDINT := UDINT#16#F2FD; (* < 62205 - HVESP22S1 *)
    PGN_HIGH_VOLTAGE_ENERGY_STORAGE_PACK_22_DATA_7 : UDINT := UDINT#16#F2FE; (* < 62206 - HVESP22D7 *)
    PGN_HIGH_VOLTAGE_ENERGY_STORAGE_PACK_22_MODULE_STATUS_1 : UDINT := UDINT#16#F2FF; (* < 62207 - HVESP22MS1 *)
    PGN_HIGH_VOLTAGE_ENERGY_STORAGE_PACK_22_THERMAL_MANAGEMENT_SYSTEM_STATUS_1 : UDINT := UDINT#16#F300; (* < 62208 - HVESP22TS1 *)
    PGN_HIGH_VOLTAGE_ENERGY_STORAGE_PACK_22_DATA_8 : UDINT := UDINT#16#F301; (* < 62209 - HVESP22D8 *)
    PGN_HIGH_VOLTAGE_ENERGY_STORAGE_PACK_22_DATA_9 : UDINT := UDINT#16#F302; (* < 62210 - HVESP22D9 *)
    PGN_HIGH_VOLTAGE_ENERGY_STORAGE_PACK_22_DATA_10 : UDINT := UDINT#16#F303; (* < 62211 - HVESP22D10 *)
    PGN_HIGH_VOLTAGE_ENERGY_STORAGE_PACK_22_DATA_11 : UDINT := UDINT#16#F304; (* < 62212 - HVESP22D11 *)
    PGN_HIGH_VOLTAGE_ENERGY_STORAGE_PACK_23_STATUS_2 : UDINT := UDINT#16#F305; (* < 62213 - HVESP23S2 *)
    PGN_HIGH_VOLTAGE_ENERGY_STORAGE_PACK_23_DATA_1 : UDINT := UDINT#16#F306; (* < 62214 - HVESP23D1 *)
    PGN_HIGH_VOLTAGE_ENERGY_STORAGE_PACK_23_DATA_2 : UDINT := UDINT#16#F307; (* < 62215 - HVESP23D2 *)
    PGN_HIGH_VOLTAGE_ENERGY_STORAGE_PACK_23_DATA_3 : UDINT := UDINT#16#F308; (* < 62216 - HVESP23D3 *)
    PGN_HIGH_VOLTAGE_ENERGY_STORAGE_PACK_23_DATA_4 : UDINT := UDINT#16#F309; (* < 62217 - HVESP23D4 *)
    PGN_HIGH_VOLTAGE_ENERGY_STORAGE_PACK_23_DATA_5 : UDINT := UDINT#16#F30A; (* < 62218 - HVESP23D5 *)
    PGN_HIGH_VOLTAGE_ENERGY_STORAGE_PACK_23_DATA_6 : UDINT := UDINT#16#F30B; (* < 62219 - HVESP23D6 *)
    PGN_HIGH_VOLTAGE_ENERGY_STORAGE_PACK_23_STATUS_1 : UDINT := UDINT#16#F30C; (* < 62220 - HVESP23S1 *)
    PGN_HIGH_VOLTAGE_ENERGY_STORAGE_PACK_23_DATA_7 : UDINT := UDINT#16#F30D; (* < 62221 - HVESP23D7 *)
    PGN_HIGH_VOLTAGE_ENERGY_STORAGE_PACK_23_MODULE_STATUS_1 : UDINT := UDINT#16#F30E; (* < 62222 - HVESP23MS1 *)
    PGN_HIGH_VOLTAGE_ENERGY_STORAGE_PACK_23_THERMAL_MANAGEMENT_SYSTEM_STATUS_1 : UDINT := UDINT#16#F30F; (* < 62223 - HVESP23TS1 *)
    PGN_HIGH_VOLTAGE_ENERGY_STORAGE_PACK_23_DATA_8 : UDINT := UDINT#16#F310; (* < 62224 - HVESP23D8 *)
    PGN_HIGH_VOLTAGE_ENERGY_STORAGE_PACK_23_DATA_9 : UDINT := UDINT#16#F311; (* < 62225 - HVESP23D9 *)
    PGN_HIGH_VOLTAGE_ENERGY_STORAGE_PACK_23_DATA_10 : UDINT := UDINT#16#F312; (* < 62226 - HVESP23D10 *)
    PGN_HIGH_VOLTAGE_ENERGY_STORAGE_PACK_23_DATA_11 : UDINT := UDINT#16#F313; (* < 62227 - HVESP23D11 *)
    PGN_HIGH_VOLTAGE_ENERGY_STORAGE_PACK_24_STATUS_2 : UDINT := UDINT#16#F314; (* < 62228 - HVESP24S2 *)
    PGN_HIGH_VOLTAGE_ENERGY_STORAGE_PACK_24_DATA_1 : UDINT := UDINT#16#F315; (* < 62229 - HVESP24D1 *)
    PGN_HIGH_VOLTAGE_ENERGY_STORAGE_PACK_24_DATA_2 : UDINT := UDINT#16#F316; (* < 62230 - HVESP24D2 *)
    PGN_HIGH_VOLTAGE_ENERGY_STORAGE_PACK_24_DATA_3 : UDINT := UDINT#16#F317; (* < 62231 - HVESP24D3 *)
    PGN_HIGH_VOLTAGE_ENERGY_STORAGE_PACK_24_DATA_4 : UDINT := UDINT#16#F318; (* < 62232 - HVESP24D4 *)
    PGN_HIGH_VOLTAGE_ENERGY_STORAGE_PACK_24_DATA_5 : UDINT := UDINT#16#F319; (* < 62233 - HVESP24D5 *)
    PGN_HIGH_VOLTAGE_ENERGY_STORAGE_PACK_24_DATA_6 : UDINT := UDINT#16#F31A; (* < 62234 - HVESP24D6 *)
    PGN_HIGH_VOLTAGE_ENERGY_STORAGE_PACK_24_STATUS_1 : UDINT := UDINT#16#F31B; (* < 62235 - HVESP24S1 *)
    PGN_HIGH_VOLTAGE_ENERGY_STORAGE_PACK_24_DATA_7 : UDINT := UDINT#16#F31C; (* < 62236 - HVESP24D7 *)
    PGN_HIGH_VOLTAGE_ENERGY_STORAGE_PACK_24_MODULE_STATUS_1 : UDINT := UDINT#16#F31D; (* < 62237 - HVESP24MS1 *)
    PGN_HIGH_VOLTAGE_ENERGY_STORAGE_PACK_24_THERMAL_MANAGEMENT_SYSTEM_STATUS_1 : UDINT := UDINT#16#F31E; (* < 62238 - HVESP24TS1 *)
    PGN_HIGH_VOLTAGE_ENERGY_STORAGE_PACK_24_DATA_8 : UDINT := UDINT#16#F31F; (* < 62239 - HVESP24D8 *)
    PGN_HIGH_VOLTAGE_ENERGY_STORAGE_PACK_24_DATA_9 : UDINT := UDINT#16#F320; (* < 62240 - HVESP24D9 *)
    PGN_HIGH_VOLTAGE_ENERGY_STORAGE_PACK_24_DATA_10 : UDINT := UDINT#16#F321; (* < 62241 - HVESP24D10 *)
    PGN_HIGH_VOLTAGE_ENERGY_STORAGE_PACK_24_DATA_11 : UDINT := UDINT#16#F322; (* < 62242 - HVESP24D11 *)
    PGN_HIGH_VOLTAGE_ENERGY_STORAGE_PACK_25_STATUS_2 : UDINT := UDINT#16#F323; (* < 62243 - HVESP25S2 *)
    PGN_HIGH_VOLTAGE_ENERGY_STORAGE_PACK_25_DATA_1 : UDINT := UDINT#16#F324; (* < 62244 - HVESP25D1 *)
    PGN_HIGH_VOLTAGE_ENERGY_STORAGE_PACK_25_DATA_2 : UDINT := UDINT#16#F325; (* < 62245 - HVESP25D2 *)
    PGN_HIGH_VOLTAGE_ENERGY_STORAGE_PACK_25_DATA_3 : UDINT := UDINT#16#F326; (* < 62246 - HVESP25D3 *)
    PGN_HIGH_VOLTAGE_ENERGY_STORAGE_PACK_25_DATA_4 : UDINT := UDINT#16#F327; (* < 62247 - HVESP25D4 *)
    PGN_HIGH_VOLTAGE_ENERGY_STORAGE_PACK_25_DATA_5 : UDINT := UDINT#16#F328; (* < 62248 - HVESP25D5 *)
    PGN_HIGH_VOLTAGE_ENERGY_STORAGE_PACK_25_DATA_6 : UDINT := UDINT#16#F329; (* < 62249 - HVESP25D6 *)
    PGN_HIGH_VOLTAGE_ENERGY_STORAGE_PACK_25_STATUS_1 : UDINT := UDINT#16#F32A; (* < 62250 - HVESP25S1 *)
    PGN_HIGH_VOLTAGE_ENERGY_STORAGE_PACK_25_DATA_7 : UDINT := UDINT#16#F32B; (* < 62251 - HVESP25D7 *)
    PGN_HIGH_VOLTAGE_ENERGY_STORAGE_PACK_25_MODULE_STATUS_1 : UDINT := UDINT#16#F32C; (* < 62252 - HVESP25MS1 *)
    PGN_HIGH_VOLTAGE_ENERGY_STORAGE_PACK_25_THERMAL_MANAGEMENT_SYSTEM_STATUS_1 : UDINT := UDINT#16#F32D; (* < 62253 - HVESP25TS1 *)
    PGN_HIGH_VOLTAGE_ENERGY_STORAGE_PACK_25_DATA_8 : UDINT := UDINT#16#F32E; (* < 62254 - HVESP25D8 *)
    PGN_HIGH_VOLTAGE_ENERGY_STORAGE_PACK_25_DATA_9 : UDINT := UDINT#16#F32F; (* < 62255 - HVESP25D9 *)
    PGN_HIGH_VOLTAGE_ENERGY_STORAGE_PACK_25_DATA_10 : UDINT := UDINT#16#F330; (* < 62256 - HVESP25D10 *)
    PGN_HIGH_VOLTAGE_ENERGY_STORAGE_PACK_25_DATA_11 : UDINT := UDINT#16#F331; (* < 62257 - HVESP25D11 *)
    PGN_HIGH_VOLTAGE_ENERGY_STORAGE_PACK_26_STATUS_2 : UDINT := UDINT#16#F332; (* < 62258 - HVESP26S2 *)
    PGN_HIGH_VOLTAGE_ENERGY_STORAGE_PACK_26_DATA_1 : UDINT := UDINT#16#F333; (* < 62259 - HVESP26D1 *)
    PGN_HIGH_VOLTAGE_ENERGY_STORAGE_PACK_26_DATA_2 : UDINT := UDINT#16#F334; (* < 62260 - HVESP26D2 *)
    PGN_HIGH_VOLTAGE_ENERGY_STORAGE_PACK_26_DATA_3 : UDINT := UDINT#16#F335; (* < 62261 - HVESP26D3 *)
    PGN_HIGH_VOLTAGE_ENERGY_STORAGE_PACK_26_DATA_4 : UDINT := UDINT#16#F336; (* < 62262 - HVESP26D4 *)
    PGN_HIGH_VOLTAGE_ENERGY_STORAGE_PACK_26_DATA_5 : UDINT := UDINT#16#F337; (* < 62263 - HVESP26D5 *)
    PGN_HIGH_VOLTAGE_ENERGY_STORAGE_PACK_26_DATA_6 : UDINT := UDINT#16#F338; (* < 62264 - HVESP26D6 *)
    PGN_HIGH_VOLTAGE_ENERGY_STORAGE_PACK_26_STATUS_1 : UDINT := UDINT#16#F339; (* < 62265 - HVESP26S1 *)
    PGN_HIGH_VOLTAGE_ENERGY_STORAGE_PACK_26_DATA_7 : UDINT := UDINT#16#F33A; (* < 62266 - HVESP26D7 *)
    PGN_HIGH_VOLTAGE_ENERGY_STORAGE_PACK_26_MODULE_STATUS_1 : UDINT := UDINT#16#F33B; (* < 62267 - HVESP26MS1 *)
    PGN_HIGH_VOLTAGE_ENERGY_STORAGE_PACK_26_THERMAL_MANAGEMENT_SYSTEM_STATUS_1 : UDINT := UDINT#16#F33C; (* < 62268 - HVESP26TS1 *)
    PGN_HIGH_VOLTAGE_ENERGY_STORAGE_PACK_26_DATA_8 : UDINT := UDINT#16#F33D; (* < 62269 - HVESP26D8 *)
    PGN_HIGH_VOLTAGE_ENERGY_STORAGE_PACK_26_DATA_9 : UDINT := UDINT#16#F33E; (* < 62270 - HVESP26D9 *)
    PGN_HIGH_VOLTAGE_ENERGY_STORAGE_PACK_26_DATA_10 : UDINT := UDINT#16#F33F; (* < 62271 - HVESP26D10 *)
    PGN_HIGH_VOLTAGE_ENERGY_STORAGE_PACK_26_DATA_11 : UDINT := UDINT#16#F340; (* < 62272 - HVESP26D11 *)
    PGN_EXTERNAL_STEERING_REQUEST : UDINT := UDINT#16#F341; (* < 62273 - XSR *)
    PGN_ACTIVE_STEERING_SYSTEM_CONTROLLER_2 : UDINT := UDINT#16#F342; (* < 62274 - ASSC2 *)
    PGN_ELECTRONIC_PARK_BRAKE_CONTROLLER_1 : UDINT := UDINT#16#F343; (* < 62275 - EPBC1 *)
    PGN_ELECTRONIC_PARK_BRAKE_CONTROLLER_2 : UDINT := UDINT#16#F344; (* < 62276 - EPBC2 *)
    PGN_GENSET_FREQUENCY_LIMITATION : UDINT := UDINT#16#F345; (* < 62277 - GFL *)
    PGN_GENSET_POWER_LIMITATION : UDINT := UDINT#16#F346; (* < 62278 - GPL *)
    PGN_GENSET_REAL_POWER_CONTROL : UDINT := UDINT#16#F347; (* < 62279 - GRPC *)
    PGN_GENSET_REACTIVE_POWER : UDINT := UDINT#16#F348; (* < 62280 - GRP *)
